C01810=1184.389,279.938,-67.679,-176.938,7.454,148.522
C01811=1184.393,279.690,-67.650,-176.940,7.452,148.522
C01812=1184.397,279.442,-67.621,-176.943,7.449,148.522
C01813=1184.402,279.194,-67.592,-176.946,7.446,148.522
C01814=1184.406,278.945,-67.564,-176.949,7.443,148.522
C01815=1184.410,278.696,-67.535,-176.951,7.441,148.523
C01816=1184.415,278.449,-67.506,-176.954,7.438,148.523
C01817=1184.419,278.200,-67.478,-176.957,7.435,148.523
C01818=1184.423,277.951,-67.449,-176.959,7.433,148.523
C01819=1184.428,277.704,-67.420,-176.962,7.430,148.523
C01820=1184.432,277.455,-67.392,-176.964,7.427,148.523
C01821=1184.437,277.207,-67.364,-176.967,7.425,148.523
C01822=1184.441,276.959,-67.335,-176.969,7.422,148.523
C01823=1184.445,276.710,-67.306,-176.972,7.419,148.523
C01824=1184.450,276.462,-67.278,-176.975,7.416,148.523
C01825=1184.454,276.214,-67.250,-176.977,7.413,148.523
C01826=1184.458,275.965,-67.220,-176.980,7.410,148.523
C01827=1184.462,275.717,-67.192,-176.982,7.407,148.523
C01828=1184.467,275.469,-67.164,-176.985,7.406,148.523
C01829=1184.471,275.221,-67.136,-176.988,7.403,148.523
C01830=1184.476,274.972,-67.107,-176.990,7.400,148.523
C01831=1184.480,274.724,-67.079,-176.993,7.398,148.524
C01832=1184.484,274.476,-67.050,-176.995,7.395,148.524
C01833=1184.488,274.227,-67.022,-176.998,7.392,148.524
C01834=1184.493,273.979,-66.993,-177.000,7.389,148.524
C01835=1184.497,273.730,-66.965,-177.003,7.386,148.524
C01836=1184.502,273.482,-66.937,-177.006,7.383,148.524
C01837=1184.506,273.233,-66.909,-177.008,7.381,148.524
C01838=1184.511,272.985,-66.880,-177.011,7.379,148.524
C01839=1184.515,272.737,-66.852,-177.014,7.376,148.524
C01840=1184.520,272.489,-66.824,-177.016,7.373,148.524
C01841=1184.523,272.241,-66.795,-177.019,7.370,148.524
C01842=1184.528,271.992,-66.766,-177.021,7.367,148.524
C01843=1184.532,271.744,-66.738,-177.023,7.365,148.524
C01844=1184.536,271.495,-66.710,-177.026,7.362,148.524
C01845=1184.541,271.247,-66.682,-177.029,7.359,148.525
C01846=1184.544,270.998,-66.654,-177.031,7.357,148.525
C01847=1184.550,270.750,-66.625,-177.034,7.354,148.525
C01848=1184.554,270.501,-66.598,-177.037,7.352,148.525
C01849=1184.559,270.253,-66.570,-177.039,7.349,148.525
C01850=1184.562,270.004,-66.541,-177.042,7.346,148.525
C01851=1184.567,269.756,-66.514,-177.045,7.343,148.525
C01852=1184.572,269.508,-66.485,-177.047,7.341,148.525
C01853=1184.576,269.260,-66.457,-177.049,7.338,148.525
C01854=1184.580,269.012,-66.429,-177.052,7.336,148.526
C01855=1184.584,268.763,-66.401,-177.055,7.333,148.526
C01856=1184.589,268.515,-66.373,-177.058,7.330,148.526
C01857=1184.593,268.266,-66.345,-177.060,7.328,148.526
C01858=1184.598,268.018,-66.317,-177.062,7.325,148.526
C01859=1184.602,267.769,-66.289,-177.065,7.322,148.526
C01860=1184.606,267.521,-66.261,-177.068,7.320,148.526
C01861=1184.611,267.273,-66.233,-177.071,7.317,148.526
C01862=1184.615,267.024,-66.205,-177.073,7.314,148.526
C01863=1184.620,266.776,-66.178,-177.075,7.312,148.526
C01864=1184.623,266.527,-66.149,-177.078,7.309,148.526
C01865=1184.628,266.279,-66.121,-177.080,7.307,148.526
C01866=1184.632,266.030,-66.094,-177.084,7.305,148.527
C01867=1184.637,265.782,-66.066,-177.086,7.302,148.527
C01868=1184.641,265.534,-66.038,-177.088,7.299,148.527
C01869=1184.646,265.285,-66.009,-177.091,7.296,148.527
C01870=1184.650,265.037,-65.982,-177.094,7.293,148.527
C01871=1184.655,264.789,-65.954,-177.096,7.291,148.527
C01872=1184.658,264.540,-65.926,-177.099,7.289,148.527
C01873=1184.664,264.292,-65.899,-177.101,7.286,148.527
C01874=1184.668,264.043,-65.871,-177.104,7.283,148.527
C01875=1184.672,263.795,-65.843,-177.107,7.280,148.527
C01876=1184.677,263.547,-65.816,-177.109,7.278,148.528
C01877=1184.680,263.298,-65.788,-177.112,7.276,148.528
C01878=1184.685,263.050,-65.761,-177.114,7.273,148.528
C01879=1184.690,262.777,-65.730,-177.117,7.270,148.528
C01880=1184.695,262.504,-65.700,-177.120,7.268,148.528
C01881=1184.700,262.231,-65.669,-177.123,7.265,148.528
C01882=1184.705,261.958,-65.639,-177.126,7.262,148.528
C01883=1184.709,261.710,-65.611,-177.129,7.259,148.528
C01884=1184.713,261.461,-65.583,-177.131,7.257,148.529
C01885=1184.718,261.213,-65.556,-177.134,7.254,148.529
C01886=1184.722,260.964,-65.528,-177.137,7.251,148.529
C01887=1184.727,260.716,-65.501,-177.139,7.249,148.529
C01888=1184.731,260.467,-65.473,-177.142,7.246,148.529
C01889=1184.735,260.219,-65.446,-177.144,7.244,148.529
C01890=1184.740,259.971,-65.418,-177.147,7.241,148.529
C01891=1184.744,259.722,-65.391,-177.149,7.239,148.529
C01892=1184.748,259.474,-65.363,-177.152,7.236,148.529
C01893=1184.753,259.225,-65.336,-177.155,7.233,148.530
C01894=1184.757,258.977,-65.309,-177.157,7.231,148.530
C01895=1184.761,258.728,-65.281,-177.160,7.228,148.530
C01896=1184.766,258.480,-65.254,-177.162,7.226,148.530
C01897=1184.770,258.231,-65.227,-177.165,7.223,148.530
C01898=1184.775,257.983,-65.199,-177.167,7.221,148.530
C01899=1184.779,257.734,-65.172,-177.170,7.218,148.530
C01900=1184.783,257.486,-65.145,-177.173,7.216,148.531
C01901=1184.788,257.238,-65.117,-177.175,7.213,148.531
C01902=1184.793,256.989,-65.090,-177.178,7.210,148.531
C01903=1184.797,256.740,-65.062,-177.180,7.208,148.531
C01904=1184.801,256.492,-65.035,-177.184,7.206,148.531
C01905=1184.806,256.244,-65.007,-177.186,7.203,148.531
C01906=1184.810,255.995,-64.980,-177.188,7.200,148.531
C01907=1184.815,255.747,-64.953,-177.191,7.197,148.531
C01908=1184.819,255.497,-64.926,-177.194,7.196,148.532
C01909=1184.823,255.250,-64.899,-177.197,7.193,148.532
C01910=1184.827,255.001,-64.872,-177.199,7.191,148.532
C01911=1184.832,254.753,-64.845,-177.202,7.188,148.532
C01912=1184.837,254.504,-64.818,-177.204,7.186,148.532
C01913=1184.841,254.256,-64.791,-177.207,7.183,148.532
C01914=1184.845,254.007,-64.763,-177.209,7.181,148.532
C01915=1184.850,253.758,-64.736,-177.212,7.178,148.533
C01916=1184.855,253.510,-64.709,-177.214,7.176,148.533
C01917=1184.858,253.262,-64.682,-177.217,7.173,148.533
C01918=1184.863,253.014,-64.655,-177.220,7.171,148.533
C01919=1184.867,252.765,-64.628,-177.222,7.168,148.533
C01920=1184.872,252.517,-64.601,-177.225,7.165,148.533
C01921=1184.876,252.267,-64.573,-177.228,7.163,148.533
C01922=1184.880,252.019,-64.547,-177.231,7.160,148.533
C01923=1184.885,251.771,-64.520,-177.233,7.158,148.534
C01924=1184.889,251.522,-64.493,-177.236,7.155,148.534
C01925=1184.894,251.274,-64.466,-177.238,7.153,148.534
C01926=1184.898,251.026,-64.439,-177.241,7.150,148.534
C01927=1184.903,250.777,-64.412,-177.243,7.148,148.534
C01928=1184.907,250.529,-64.385,-177.246,7.145,148.534
C01929=1184.912,250.280,-64.358,-177.248,7.143,148.534
C01930=1184.915,250.031,-64.331,-177.252,7.141,148.535
C01931=1184.920,249.783,-64.304,-177.254,7.138,148.535
C01932=1184.925,249.534,-64.278,-177.256,7.135,148.535
C01933=1184.930,249.285,-64.251,-177.259,7.134,148.535
C01934=1184.933,249.037,-64.224,-177.262,7.131,148.535
C01935=1184.938,248.788,-64.197,-177.264,7.129,148.535
C01936=1184.943,248.540,-64.170,-177.267,7.126,148.536
C01937=1184.947,248.292,-64.144,-177.269,7.124,148.536
C01938=1184.951,248.043,-64.116,-177.272,7.121,148.536
C01939=1184.956,247.794,-64.090,-177.275,7.119,148.536
C01940=1184.960,247.546,-64.064,-177.278,7.116,148.536
C01941=1184.965,247.298,-64.037,-177.280,7.114,148.536
C01942=1184.969,247.049,-64.010,-177.283,7.111,148.537
C01943=1184.973,246.801,-63.983,-177.285,7.109,148.537
C01944=1184.978,246.552,-63.957,-177.288,7.106,148.537
C01945=1184.982,246.304,-63.930,-177.290,7.104,148.537
C01946=1184.987,246.055,-63.903,-177.293,7.101,148.537
C01947=1184.991,245.806,-63.877,-177.296,7.099,148.537
C01948=1184.996,245.558,-63.850,-177.299,7.096,148.537
C01949=1185.001,245.309,-63.823,-177.301,7.094,148.538
C01950=1185.004,245.061,-63.797,-177.304,7.092,148.538
C01951=1185.009,244.812,-63.770,-177.306,7.089,148.538
C01952=1185.013,244.564,-63.744,-177.309,7.088,148.538
C01953=1185.018,244.315,-63.717,-177.311,7.085,148.538
C01954=1185.022,244.066,-63.691,-177.314,7.082,148.538
C01955=1185.027,243.818,-63.664,-177.317,7.080,148.539
C01956=1185.031,243.569,-63.638,-177.319,7.078,148.539
C01957=1185.036,243.321,-63.611,-177.322,7.075,148.539
C01958=1185.040,243.072,-63.585,-177.324,7.073,148.539
C01959=1185.045,242.823,-63.559,-177.327,7.070,148.539
C01960=1185.049,242.575,-63.532,-177.330,7.068,148.540
C01961=1185.054,242.326,-63.506,-177.333,7.065,148.540
C01962=1185.057,242.078,-63.479,-177.335,7.063,148.540
C01963=1185.062,241.829,-63.453,-177.338,7.060,148.540
C01964=1185.067,241.581,-63.427,-177.341,7.058,148.540
C01965=1185.072,241.332,-63.400,-177.343,7.056,148.540
C01966=1185.076,241.084,-63.374,-177.345,7.053,148.540
C01967=1185.081,240.835,-63.348,-177.348,7.052,148.541
C01968=1185.085,240.587,-63.321,-177.351,7.049,148.541
C01969=1185.089,240.338,-63.295,-177.353,7.047,148.541
C01970=1185.094,240.089,-63.268,-177.356,7.044,148.541
C01971=1185.098,239.841,-63.243,-177.359,7.042,148.542
C01972=1185.102,239.592,-63.216,-177.362,7.039,148.542
C01973=1185.107,239.344,-63.190,-177.364,7.037,148.542
C01974=1185.112,239.095,-63.164,-177.366,7.035,148.542
C01975=1185.116,238.847,-63.137,-177.369,7.032,148.542
C01976=1185.120,238.598,-63.112,-177.372,7.030,148.542
C01977=1185.125,238.349,-63.086,-177.375,7.027,148.543
C01978=1185.129,238.101,-63.059,-177.377,7.025,148.543
C01979=1185.134,237.852,-63.033,-177.380,7.022,148.543
C01980=1185.138,237.604,-63.008,-177.383,7.021,148.543
C01981=1185.143,237.355,-62.981,-177.385,7.018,148.543
C01982=1185.147,237.106,-62.955,-177.388,7.016,148.544
C01983=1185.152,236.835,-62.926,-177.391,7.013,148.544
C01984=1185.157,236.563,-62.897,-177.393,7.011,148.544
C01985=1185.162,236.292,-62.870,-177.397,7.008,148.544
C01986=1185.167,236.020,-62.841,-177.399,7.005,148.544
C01987=1185.171,235.772,-62.815,-177.402,7.004,148.545
C01988=1185.176,235.522,-62.789,-177.404,7.001,148.545
C01989=1185.180,235.274,-62.762,-177.407,6.999,148.545
C01990=1185.185,235.026,-62.737,-177.409,6.997,148.545
C01991=1185.189,234.777,-62.711,-177.413,6.994,148.545
C01992=1185.194,234.528,-62.685,-177.415,6.992,148.546
C01993=1185.198,234.279,-62.659,-177.418,6.989,148.546
C01994=1185.202,234.031,-62.633,-177.420,6.987,148.546
C01995=1185.207,233.783,-62.607,-177.423,6.985,148.546
C01996=1185.211,233.534,-62.582,-177.426,6.982,148.546
C01997=1185.216,233.285,-62.555,-177.428,6.980,148.547
C01998=1185.220,233.036,-62.530,-177.430,6.978,148.547
C01999=1185.225,232.788,-62.504,-177.434,6.976,148.547
C02000=1185.229,232.540,-62.478,-177.436,6.974,148.547
C02001=1185.233,232.291,-62.453,-177.439,6.971,148.547
C02002=1185.238,232.043,-62.427,-177.441,6.969,148.548
C02003=1185.243,231.794,-62.401,-177.444,6.967,148.548
C02004=1185.247,231.545,-62.375,-177.447,6.964,148.548
C02005=1185.252,231.296,-62.349,-177.449,6.962,148.548
C02006=1185.257,231.048,-62.324,-177.452,6.959,148.548
C02007=1185.261,230.799,-62.298,-177.455,6.957,148.549
C02008=1185.265,230.550,-62.273,-177.457,6.955,148.549
C02009=1185.270,230.302,-62.247,-177.460,6.953,148.549
C02010=1185.274,230.053,-62.221,-177.463,6.951,148.549
C02011=1185.278,229.804,-62.196,-177.465,6.949,148.550
C02012=1185.282,229.556,-62.170,-177.468,6.946,148.550
C02013=1185.287,229.308,-62.144,-177.470,6.944,148.550
C02014=1185.292,229.059,-62.119,-177.473,6.942,148.550
C02015=1185.297,228.810,-62.092,-177.476,6.939,148.550
C02016=1185.301,228.562,-62.067,-177.478,6.937,148.551
C02017=1185.306,228.312,-62.042,-177.481,6.934,148.551
C02018=1185.311,228.064,-62.017,-177.484,6.932,148.551
C02019=1185.315,227.815,-61.991,-177.486,6.931,148.551
C02020=1185.319,227.566,-61.965,-177.489,6.928,148.551
C02021=1185.324,227.318,-61.940,-177.492,6.926,148.552
C02022=1185.328,227.069,-61.914,-177.494,6.924,148.552
C02023=1185.333,226.820,-61.889,-177.497,6.921,148.552
C02024=1185.338,226.572,-61.864,-177.499,6.919,148.552
C02025=1185.342,226.323,-61.838,-177.502,6.917,148.553
C02026=1185.346,226.074,-61.812,-177.505,6.914,148.553
C02027=1185.350,225.827,-61.787,-177.507,6.912,148.553
C02028=1185.355,225.577,-61.762,-177.510,6.910,148.553
C02029=1185.359,225.329,-61.737,-177.513,6.907,148.553
C02030=1185.364,225.080,-61.711,-177.515,6.906,148.554
C02031=1185.368,224.831,-61.686,-177.518,6.904,148.554
C02032=1185.373,224.583,-61.661,-177.521,6.901,148.554
C02033=1185.377,224.334,-61.635,-177.523,6.899,148.555
C02034=1185.382,224.085,-61.610,-177.526,6.897,148.555
C02035=1185.387,223.836,-61.584,-177.529,6.894,148.555
C02036=1185.391,223.588,-61.559,-177.531,6.892,148.555
C02037=1185.396,223.339,-61.534,-177.534,6.890,148.555
C02038=1185.400,223.091,-61.509,-177.537,6.888,148.556
C02039=1185.404,222.842,-61.484,-177.539,6.886,148.556
C02040=1185.409,222.593,-61.458,-177.542,6.884,148.556
C02041=1185.414,222.345,-61.433,-177.545,6.881,148.556
C02042=1185.418,222.095,-61.408,-177.547,6.879,148.557
C02043=1185.423,221.847,-61.383,-177.550,6.877,148.557
C02044=1185.426,221.599,-61.358,-177.552,6.874,148.557
C02045=1185.432,221.350,-61.333,-177.555,6.872,148.557
C02046=1185.436,221.101,-61.307,-177.558,6.871,148.558
C02047=1185.441,220.852,-61.282,-177.560,6.868,148.558
C02048=1185.445,220.604,-61.257,-177.563,6.866,148.558
C02049=1185.450,220.355,-61.233,-177.566,6.864,148.558
C02050=1185.454,220.106,-61.207,-177.568,6.862,148.558
C02051=1185.459,219.858,-61.182,-177.571,6.859,148.559
C02052=1185.463,219.609,-61.156,-177.574,6.857,148.559
C02053=1185.468,219.360,-61.132,-177.576,6.855,148.559
C02054=1185.472,219.111,-61.107,-177.579,6.853,148.560
C02055=1185.477,218.863,-61.082,-177.582,6.851,148.560
C02056=1185.481,218.614,-61.057,-177.584,6.849,148.560
C02057=1185.486,218.366,-61.032,-177.587,6.846,148.560
C02058=1185.490,218.116,-61.007,-177.589,6.844,148.560
C02059=1185.495,217.868,-60.982,-177.592,6.842,148.561
C02060=1185.499,217.620,-60.958,-177.595,6.840,148.561
C02061=1185.504,217.370,-60.933,-177.598,6.837,148.561
C02062=1185.509,217.122,-60.908,-177.600,6.835,148.561
C02063=1185.512,216.873,-60.883,-177.603,6.834,148.562
C02064=1185.518,216.624,-60.858,-177.606,6.831,148.562
C02065=1185.522,216.375,-60.833,-177.608,6.829,148.562
C02066=1185.526,216.127,-60.808,-177.611,6.827,148.563
C02067=1185.531,215.878,-60.784,-177.613,6.825,148.563
C02068=1185.536,215.629,-60.759,-177.616,6.822,148.563
C02069=1185.540,215.381,-60.734,-177.619,6.820,148.563
C02070=1185.544,215.132,-60.709,-177.622,6.819,148.564
C02071=1185.549,214.883,-60.685,-177.624,6.816,148.564
C02072=1185.554,214.635,-60.660,-177.627,6.814,148.564
C02073=1185.559,214.385,-60.635,-177.630,6.812,148.564
C02074=1185.563,214.137,-60.610,-177.632,6.810,148.565
C02075=1185.567,213.888,-60.585,-177.635,6.807,148.565
C02076=1185.572,213.640,-60.561,-177.638,6.806,148.565
C02077=1185.577,213.391,-60.536,-177.640,6.803,148.565
C02078=1185.580,213.142,-60.512,-177.643,6.802,148.566
C02079=1185.586,212.893,-60.487,-177.646,6.799,148.566
C02080=1185.590,212.645,-60.462,-177.648,6.797,148.566
C02081=1185.594,212.396,-60.437,-177.651,6.795,148.566
C02082=1185.599,212.147,-60.413,-177.653,6.793,148.567
C02083=1185.604,211.899,-60.389,-177.656,6.791,148.567
C02084=1185.608,211.649,-60.364,-177.659,6.788,148.567
C02085=1185.613,211.401,-60.340,-177.661,6.787,148.568
C02086=1185.618,211.152,-60.315,-177.664,6.785,148.568
C02087=1185.622,210.882,-60.288,-177.667,6.782,148.568
C02088=1185.627,210.611,-60.262,-177.669,6.780,148.568
C02089=1185.632,210.341,-60.235,-177.673,6.777,148.569
C02090=1185.637,210.070,-60.209,-177.676,6.775,148.569
C02091=1185.641,209.821,-60.185,-177.678,6.773,148.569
C02092=1185.646,209.573,-60.160,-177.681,6.771,148.570
C02093=1185.651,209.324,-60.136,-177.683,6.769,148.570
C02094=1185.655,209.075,-60.111,-177.686,6.767,148.570
C02095=1185.660,208.826,-60.087,-177.689,6.765,148.570
C02096=1185.665,208.578,-60.062,-177.692,6.763,148.571
C02097=1185.669,208.329,-60.038,-177.694,6.761,148.571
C02098=1185.673,208.080,-60.014,-177.697,6.759,148.571
C02099=1185.678,207.831,-59.989,-177.700,6.756,148.571
C02100=1185.682,207.583,-59.965,-177.703,6.754,148.572
C02101=1185.688,207.334,-59.940,-177.705,6.752,148.572
C02102=1185.691,207.085,-59.916,-177.707,6.750,148.572
C02103=1185.696,206.836,-59.892,-177.710,6.749,148.573
C02104=1185.701,206.587,-59.868,-177.713,6.746,148.573
C02105=1185.706,206.339,-59.844,-177.716,6.744,148.573
C02106=1185.709,206.090,-59.819,-177.718,6.742,148.573
C02107=1185.715,205.841,-59.794,-177.721,6.740,148.574
C02108=1185.719,205.592,-59.771,-177.724,6.737,148.574
C02109=1185.724,205.344,-59.747,-177.726,6.736,148.574
C02110=1185.729,205.095,-59.722,-177.729,6.734,148.574
C02111=1185.733,204.846,-59.698,-177.732,6.732,148.575
C02112=1185.737,204.597,-59.674,-177.734,6.730,148.575
C02113=1185.742,204.348,-59.651,-177.737,6.727,148.575
C02114=1185.747,204.100,-59.626,-177.740,6.725,148.576
C02115=1185.751,203.851,-59.602,-177.742,6.724,148.576
C02116=1185.755,203.602,-59.578,-177.745,6.722,148.576
C02117=1185.760,203.353,-59.554,-177.747,6.720,148.576
C02118=1185.765,203.104,-59.529,-177.750,6.717,148.577
C02119=1185.769,202.856,-59.505,-177.753,6.715,148.577
C02120=1185.774,202.607,-59.482,-177.756,6.713,148.577
C02121=1185.778,202.359,-59.458,-177.758,6.711,148.578
C02122=1185.782,202.109,-59.434,-177.761,6.709,148.578
C02123=1185.788,201.860,-59.409,-177.764,6.707,148.578
C02124=1185.792,201.612,-59.385,-177.766,6.705,148.579
C02125=1185.797,201.363,-59.362,-177.769,6.703,148.579
C02126=1185.801,201.114,-59.338,-177.771,6.701,148.579
C02127=1185.806,200.865,-59.315,-177.774,6.699,148.579
C02128=1185.811,200.617,-59.290,-177.777,6.698,148.580
C02129=1185.815,200.368,-59.266,-177.780,6.695,148.580
C02130=1185.819,200.118,-59.242,-177.782,6.693,148.580
C02131=1185.824,199.870,-59.218,-177.785,6.691,148.581
C02132=1185.828,199.621,-59.195,-177.787,6.689,148.581
C02133=1185.833,199.373,-59.171,-177.790,6.687,148.581
C02134=1185.838,199.123,-59.147,-177.793,6.686,148.582
C02135=1185.842,198.875,-59.123,-177.796,6.683,148.582
C02136=1185.847,198.626,-59.099,-177.798,6.681,148.582
C02137=1185.852,198.377,-59.075,-177.801,6.679,148.582
C02138=1185.856,198.128,-59.052,-177.803,6.677,148.583
C02139=1185.861,197.880,-59.028,-177.806,6.675,148.583
C02140=1185.866,197.631,-59.004,-177.809,6.674,148.583
C02141=1185.870,197.382,-58.981,-177.811,6.671,148.583
C02142=1185.874,197.133,-58.956,-177.814,6.669,148.584
C02143=1185.879,196.884,-58.933,-177.817,6.667,148.584
C02144=1185.883,196.635,-58.909,-177.819,6.665,148.585
C02145=1185.888,196.386,-58.886,-177.822,6.663,148.585
C02146=1185.893,196.137,-58.862,-177.825,6.662,148.585
C02147=1185.897,195.889,-58.838,-177.827,6.660,148.585
C02148=1185.902,195.640,-58.815,-177.830,6.657,148.586
C02149=1185.906,195.391,-58.792,-177.833,6.655,148.586
C02150=1185.911,195.142,-58.767,-177.836,6.653,148.586
C02151=1185.915,194.893,-58.744,-177.838,6.652,148.587
C02152=1185.920,194.644,-58.721,-177.841,6.650,148.587
C02153=1185.925,194.395,-58.697,-177.843,6.648,148.587
C02154=1185.929,194.147,-58.673,-177.846,6.646,148.588
C02155=1185.934,193.898,-58.650,-177.848,6.644,148.588
C02156=1185.939,193.649,-58.627,-177.852,6.641,148.588
C02157=1185.943,193.400,-58.603,-177.854,6.640,148.589
C02158=1185.948,193.151,-58.579,-177.857,6.638,148.589
C02159=1185.952,192.902,-58.556,-177.859,6.636,148.589
C02160=1185.957,192.653,-58.532,-177.862,6.634,148.589
C02161=1185.962,192.404,-58.509,-177.864,6.632,148.590
C02162=1185.966,192.155,-58.486,-177.867,6.630,148.590
C02163=1185.971,191.908,-58.463,-177.870,6.628,148.590
C02164=1185.975,191.659,-58.439,-177.873,6.626,148.591
C02165=1185.980,191.410,-58.416,-177.876,6.624,148.591
C02166=1185.985,191.161,-58.393,-177.878,6.622,148.591
C02167=1185.990,190.912,-58.369,-177.881,6.620,148.592
C02168=1185.994,190.663,-58.346,-177.883,6.618,148.592
C02169=1185.999,190.414,-58.322,-177.886,6.617,148.592
C02170=1186.003,190.165,-58.300,-177.889,6.615,148.593
C02171=1186.007,189.916,-58.276,-177.891,6.613,148.593
C02172=1186.012,189.667,-58.252,-177.894,6.611,148.593
C02173=1186.017,189.418,-58.229,-177.897,6.608,148.593
C02174=1186.021,189.169,-58.206,-177.899,6.606,148.594
C02175=1186.027,188.921,-58.183,-177.902,6.605,148.594
C02176=1186.031,188.672,-58.160,-177.905,6.603,148.595
C02177=1186.035,188.423,-58.136,-177.907,6.601,148.595
C02178=1186.040,188.174,-58.113,-177.910,6.599,148.595
C02179=1186.045,187.925,-58.090,-177.913,6.597,148.596
C02180=1186.049,187.676,-58.067,-177.915,6.596,148.596
C02181=1186.053,187.427,-58.044,-177.918,6.594,148.596
C02182=1186.058,187.178,-58.020,-177.920,6.592,148.596
C02183=1186.063,186.930,-57.997,-177.923,6.590,148.597
C02184=1186.067,186.681,-57.974,-177.925,6.588,148.597
C02185=1186.072,186.432,-57.952,-177.929,6.586,148.597
C02186=1186.077,186.183,-57.928,-177.931,6.584,148.598
C02187=1186.082,185.934,-57.905,-177.934,6.582,148.598
C02188=1186.086,185.685,-57.882,-177.937,6.580,148.599
C02189=1186.091,185.437,-57.859,-177.939,6.578,148.599
C02190=1186.096,185.188,-57.836,-177.942,6.577,148.599
C02191=1186.100,184.918,-57.812,-177.945,6.575,148.600
C02192=1186.106,184.648,-57.787,-177.948,6.572,148.600
C02193=1186.111,184.379,-57.761,-177.951,6.570,148.600
C02194=1186.116,184.109,-57.737,-177.953,6.569,148.601
C02195=1186.120,183.860,-57.714,-177.956,6.567,148.601
C02196=1186.125,183.611,-57.690,-177.959,6.565,148.601
C02197=1186.129,183.362,-57.668,-177.961,6.563,148.602
C02198=1186.135,183.113,-57.645,-177.964,6.561,148.602
C02199=1186.138,182.865,-57.623,-177.966,6.559,148.602
C02200=1186.143,182.616,-57.599,-177.969,6.557,148.603
C02201=1186.148,182.367,-57.576,-177.972,6.555,148.603
C02202=1186.152,182.117,-57.554,-177.975,6.553,148.603
C02203=1186.157,181.869,-57.531,-177.977,6.551,148.604
C02204=1186.161,181.620,-57.508,-177.980,6.550,148.604
C02205=1186.166,181.371,-57.485,-177.983,6.548,148.604
C02206=1186.170,181.122,-57.463,-177.985,6.546,148.605
C02207=1186.176,180.873,-57.440,-177.988,6.544,148.605
C02208=1186.181,180.624,-57.417,-177.991,6.542,148.605
C02209=1186.185,180.375,-57.394,-177.993,6.541,148.606
C02210=1186.189,180.126,-57.371,-177.996,6.539,148.606
C02211=1186.194,179.877,-57.349,-177.999,6.537,148.606
C02212=1186.199,179.628,-57.326,-178.001,6.535,148.607
C02213=1186.203,179.380,-57.303,-178.004,6.533,148.607
C02214=1186.208,179.131,-57.281,-178.006,6.531,148.607
C02215=1186.212,178.882,-57.258,-178.009,6.530,148.608
C02216=1186.217,178.632,-57.235,-178.012,6.528,148.608
C02217=1186.221,178.384,-57.213,-178.014,6.526,148.608
C02218=1186.227,178.135,-57.190,-178.017,6.524,148.609
C02219=1186.231,177.886,-57.168,-178.020,6.522,148.609
C02220=1186.236,177.637,-57.144,-178.022,6.521,148.610
C02221=1186.241,177.388,-57.123,-178.025,6.519,148.610
C02222=1186.245,177.140,-57.100,-178.028,6.517,148.610
C02223=1186.250,176.890,-57.077,-178.030,6.515,148.611
C02224=1186.254,176.642,-57.055,-178.033,6.514,148.611
C02225=1186.259,176.392,-57.032,-178.036,6.512,148.611
C02226=1186.263,176.143,-57.010,-178.038,6.510,148.612
C02227=1186.269,175.895,-56.987,-178.041,6.508,148.612
C02228=1186.273,175.645,-56.965,-178.044,6.506,148.612
C02229=1186.277,175.396,-56.942,-178.046,6.505,148.613
C02230=1186.283,175.148,-56.920,-178.049,6.503,148.613
C02231=1186.286,174.899,-56.897,-178.052,6.501,148.613
C02232=1186.292,174.650,-56.875,-178.054,6.499,148.614
C02233=1186.296,174.401,-56.853,-178.057,6.497,148.614
C02234=1186.300,174.152,-56.830,-178.060,6.496,148.615
C02235=1186.306,173.903,-56.808,-178.062,6.494,148.615
C02236=1186.310,173.654,-56.786,-178.065,6.492,148.615
C02237=1186.315,173.406,-56.763,-178.068,6.490,148.616
C02238=1186.320,173.156,-56.741,-178.071,6.489,148.616
C02239=1186.324,172.906,-56.719,-178.073,6.487,148.616
C02240=1186.329,172.658,-56.696,-178.076,6.485,148.617
C02241=1186.334,172.409,-56.674,-178.079,6.483,148.617
C02242=1186.338,172.160,-56.652,-178.081,6.481,148.617
C02243=1186.342,171.911,-56.629,-178.084,6.480,148.618
C02244=1186.347,171.663,-56.607,-178.087,6.478,148.618
C02245=1186.352,171.413,-56.585,-178.089,6.476,148.619
C02246=1186.357,171.164,-56.563,-178.092,6.474,148.619
C02247=1186.361,170.915,-56.541,-178.095,6.473,148.619
C02248=1186.366,170.666,-56.518,-178.097,6.471,148.620
C02249=1186.371,170.418,-56.496,-178.100,6.469,148.620
C02250=1186.375,170.168,-56.474,-178.103,6.467,148.620
C02251=1186.380,169.920,-56.452,-178.105,6.465,148.621
C02252=1186.384,169.670,-56.430,-178.108,6.464,148.621
C02253=1186.390,169.422,-56.407,-178.111,6.462,148.621
C02254=1186.394,169.173,-56.385,-178.113,6.460,148.622
C02255=1186.399,168.924,-56.364,-178.116,6.458,148.622
C02256=1186.403,168.675,-56.342,-178.119,6.457,148.623
C02257=1186.409,168.426,-56.319,-178.121,6.455,148.623
C02258=1186.413,168.176,-56.297,-178.124,6.453,148.623
C02259=1186.418,167.928,-56.276,-178.126,6.452,148.624
C02260=1186.422,167.678,-56.253,-178.129,6.450,148.624
C02261=1186.427,167.430,-56.232,-178.131,6.448,148.624
C02262=1186.431,167.181,-56.209,-178.134,6.447,148.625
C02263=1186.437,166.932,-56.187,-178.137,6.445,148.625
C02264=1186.441,166.683,-56.165,-178.140,6.443,148.626
C02265=1186.446,166.434,-56.143,-178.142,6.441,148.626
C02266=1186.450,166.185,-56.121,-178.145,6.440,148.626
C02267=1186.455,165.936,-56.099,-178.148,6.438,148.627
C02268=1186.459,165.687,-56.077,-178.150,6.436,148.627
C02269=1186.464,165.438,-56.056,-178.153,6.434,148.627
C02270=1186.468,165.189,-56.034,-178.156,6.432,148.628
C02271=1186.473,164.940,-56.012,-178.158,6.431,148.628
C02272=1186.478,164.691,-55.990,-178.161,6.429,148.628
C02273=1186.482,164.442,-55.968,-178.164,6.427,148.629
C02274=1186.488,164.192,-55.947,-178.166,6.425,148.629
C02275=1186.492,163.943,-55.924,-178.168,6.424,148.630
C02276=1186.497,163.695,-55.903,-178.172,6.423,148.630
C02277=1186.502,163.445,-55.881,-178.174,6.421,148.631
C02278=1186.506,163.197,-55.859,-178.177,6.419,148.631
C02279=1186.511,162.948,-55.837,-178.180,6.418,148.631
C02280=1186.516,162.699,-55.815,-178.182,6.416,148.632
C02281=1186.520,162.450,-55.794,-178.185,6.414,148.632
C02282=1186.525,162.201,-55.772,-178.188,6.412,148.632
C02283=1186.530,161.951,-55.751,-178.190,6.410,148.633
C02284=1186.535,161.703,-55.729,-178.193,6.409,148.633
C02285=1186.539,161.453,-55.707,-178.196,6.407,148.634
C02286=1186.544,161.205,-55.685,-178.198,6.406,148.634
C02287=1186.549,160.956,-55.664,-178.200,6.404,148.634
C02288=1186.553,160.706,-55.642,-178.203,6.402,148.635
C02289=1186.558,160.457,-55.621,-178.206,6.401,148.635
C02290=1186.562,160.208,-55.599,-178.209,6.399,148.635
C02291=1186.567,159.960,-55.577,-178.212,6.397,148.636
C02292=1186.572,159.711,-55.556,-178.214,6.396,148.636
C02293=1186.576,159.461,-55.534,-178.217,6.394,148.637
C02294=1186.581,159.213,-55.513,-178.220,6.392,148.637
C02295=1186.586,158.943,-55.489,-178.222,6.390,148.638
C02296=1186.591,158.674,-55.467,-178.225,6.389,148.638
C02297=1186.596,158.405,-55.443,-178.228,6.387,148.638
C02298=1186.601,158.136,-55.420,-178.231,6.385,148.639
C02299=1186.606,157.888,-55.398,-178.234,6.384,148.639
C02300=1186.611,157.638,-55.377,-178.236,6.382,148.640
C02301=1186.615,157.389,-55.355,-178.239,6.380,148.640
C02302=1186.620,157.140,-55.333,-178.242,6.378,148.640
C02303=1186.625,156.891,-55.312,-178.244,6.377,148.641
C02304=1186.630,156.643,-55.291,-178.246,6.376,148.641
C02305=1186.634,156.393,-55.270,-178.249,6.374,148.641
C02306=1186.639,156.144,-55.248,-178.252,6.372,148.642
C02307=1186.644,155.895,-55.227,-178.255,6.371,148.642
C02308=1186.648,155.646,-55.205,-178.258,6.369,148.643
C02309=1186.653,155.397,-55.184,-178.260,6.367,148.643
C02310=1186.658,155.148,-55.163,-178.263,6.365,148.644
C02311=1186.663,154.899,-55.142,-178.265,6.364,148.644
C02312=1186.667,154.649,-55.120,-178.268,6.363,148.644
C02313=1186.672,154.401,-55.099,-178.271,6.361,148.645
C02314=1186.676,154.152,-55.078,-178.273,6.359,148.645
C02315=1186.681,153.903,-55.056,-178.276,6.358,148.646
C02316=1186.686,153.653,-55.035,-178.279,6.356,148.646
C02317=1186.691,153.405,-55.013,-178.282,6.354,148.646
C02318=1186.695,153.156,-54.993,-178.284,6.353,148.647
C02319=1186.700,152.906,-54.972,-178.287,6.351,148.647
C02320=1186.705,152.658,-54.950,-178.289,6.350,148.648
C02321=1186.710,152.408,-54.929,-178.292,6.348,148.648
C02322=1186.714,152.159,-54.908,-178.295,6.346,148.648
C02323=1186.719,151.910,-54.887,-178.298,6.345,148.649
C02324=1186.724,151.662,-54.865,-178.300,6.344,148.649
C02325=1186.728,151.413,-54.845,-178.303,6.342,148.650
C02326=1186.733,151.163,-54.824,-178.305,6.340,148.650
C02327=1186.738,150.914,-54.802,-178.308,6.338,148.650
C02328=1186.742,150.665,-54.782,-178.311,6.337,148.651
C02329=1186.748,150.416,-54.761,-178.313,6.335,148.651
C02330=1186.752,150.167,-54.739,-178.316,6.334,148.652
C02331=1186.757,149.918,-54.719,-178.319,6.332,148.652
C02332=1186.761,149.668,-54.697,-178.321,6.331,148.653
C02333=1186.766,149.420,-54.676,-178.324,6.329,148.653
C02334=1186.771,149.171,-54.655,-178.327,6.327,148.653
C02335=1186.776,148.921,-54.634,-178.329,6.325,148.654
C02336=1186.781,148.672,-54.613,-178.331,6.324,148.654
C02337=1186.785,148.424,-54.592,-178.335,6.323,148.655
C02338=1186.790,148.175,-54.571,-178.337,6.321,148.655
C02339=1186.794,147.925,-54.550,-178.340,6.319,148.656
C02340=1186.799,147.676,-54.530,-178.343,6.318,148.656
C02341=1186.804,147.427,-54.508,-178.345,6.317,148.656
C02342=1186.809,147.178,-54.487,-178.347,6.315,148.657
C02343=1186.814,146.929,-54.466,-178.351,6.314,148.657
C02344=1186.818,146.680,-54.446,-178.353,6.312,148.658
C02345=1186.823,146.431,-54.425,-178.356,6.310,148.658
C02346=1186.828,146.182,-54.405,-178.359,6.308,148.658
C02347=1186.833,145.933,-54.383,-178.361,6.307,148.659
C02348=1186.837,145.684,-54.363,-178.364,6.306,148.659
C02349=1186.842,145.434,-54.341,-178.367,6.304,148.660
C02350=1186.846,145.185,-54.321,-178.369,6.302,148.660
C02351=1186.851,144.936,-54.300,-178.371,6.301,148.661
C02352=1186.856,144.687,-54.280,-178.374,6.300,148.661
C02353=1186.861,144.438,-54.259,-178.377,6.298,148.661
C02354=1186.865,144.189,-54.238,-178.380,6.296,148.662
C02355=1186.871,143.939,-54.217,-178.383,6.295,148.662
C02356=1186.875,143.691,-54.197,-178.385,6.294,148.663
C02357=1186.880,143.441,-54.176,-178.388,6.292,148.663
C02358=1186.884,143.193,-54.155,-178.390,6.290,148.664
C02359=1186.890,142.944,-54.134,-178.393,6.289,148.664
C02360=1186.894,142.695,-54.114,-178.396,6.287,148.664
C02361=1186.898,142.446,-54.093,-178.398,6.286,148.665
C02362=1186.904,142.197,-54.072,-178.401,6.284,148.665
C02363=1186.908,141.948,-54.052,-178.404,6.283,148.666
C02364=1186.914,141.698,-54.032,-178.406,6.281,148.666
C02365=1186.918,141.449,-54.011,-178.409,6.280,148.667
C02366=1186.922,141.200,-53.991,-178.412,6.279,148.667
C02367=1186.928,140.951,-53.970,-178.414,6.277,148.667
C02368=1186.932,140.702,-53.950,-178.417,6.275,148.668
C02369=1186.937,140.452,-53.929,-178.419,6.274,148.668
C02370=1186.942,140.203,-53.908,-178.422,6.273,148.669
C02371=1186.946,139.954,-53.888,-178.425,6.271,148.669
C02372=1186.951,139.705,-53.867,-178.428,6.269,148.670
C02373=1186.956,139.456,-53.847,-178.430,6.267,148.670
C02374=1186.960,139.207,-53.826,-178.432,6.266,148.670
C02375=1186.966,138.957,-53.806,-178.436,6.265,148.671
C02376=1186.970,138.708,-53.786,-178.438,6.263,148.671
C02377=1186.974,138.460,-53.765,-178.441,6.261,148.672
C02378=1186.980,138.210,-53.744,-178.443,6.261,148.672
C02379=1186.984,137.961,-53.724,-178.446,6.259,148.673
C02380=1186.988,137.712,-53.703,-178.449,6.257,148.673
C02381=1186.994,137.462,-53.683,-178.452,6.256,148.674
C02382=1186.998,137.214,-53.663,-178.454,6.255,148.674
C02383=1187.003,136.965,-53.642,-178.456,6.253,148.674
C02384=1187.007,136.716,-53.622,-178.460,6.251,148.675
C02385=1187.013,136.466,-53.602,-178.462,6.251,148.675
C02386=1187.017,136.217,-53.581,-178.464,6.249,148.676
C02387=1187.022,135.969,-53.561,-178.467,6.247,148.676
C02388=1187.027,135.720,-53.541,-178.470,6.246,148.677
C02389=1187.032,135.470,-53.521,-178.472,6.245,148.677
C02390=1187.037,135.221,-53.500,-178.475,6.243,148.678
C02391=1187.041,134.972,-53.480,-178.478,6.241,148.678
C02392=1187.046,134.722,-53.460,-178.481,6.240,148.679
C02393=1187.050,134.473,-53.440,-178.483,6.239,148.679
C02394=1187.055,134.224,-53.419,-178.486,6.237,148.679
C02395=1187.060,133.974,-53.399,-178.489,6.235,148.680
C02396=1187.065,133.726,-53.379,-178.491,6.234,148.680
C02397=1187.070,133.477,-53.359,-178.494,6.233,148.681
C02398=1187.074,133.228,-53.339,-178.496,6.231,148.681
C02399=1187.080,132.959,-53.317,-178.499,6.229,148.682
C02400=1187.085,132.691,-53.296,-178.502,6.228,148.682
C02401=1187.090,132.422,-53.274,-178.505,6.226,148.683
C02402=1187.095,132.154,-53.252,-178.508,6.225,148.683
C02403=1187.100,131.904,-53.232,-178.510,6.224,148.684
C02404=1187.105,131.655,-53.212,-178.513,6.222,148.684
C02405=1187.110,131.405,-53.192,-178.516,6.220,148.684
C02406=1187.114,131.156,-53.172,-178.518,6.220,148.685
C02407=1187.119,130.908,-53.152,-178.521,6.218,148.685
C02408=1187.124,130.659,-53.132,-178.524,6.216,148.686
C02409=1187.128,130.409,-53.112,-178.527,6.215,148.686
C02410=1187.133,130.160,-53.092,-178.529,6.214,148.687
C02411=1187.138,129.910,-53.072,-178.532,6.212,148.687
C02412=1187.143,129.662,-53.052,-178.534,6.210,148.688
C02413=1187.148,129.412,-53.032,-178.537,6.210,148.688
C02414=1187.153,129.163,-53.012,-178.540,6.208,148.689
C02415=1187.157,128.914,-52.992,-178.542,6.206,148.689
C02416=1187.162,128.665,-52.972,-178.545,6.205,148.689
C02417=1187.167,128.416,-52.952,-178.548,6.204,148.690
C02418=1187.172,128.166,-52.933,-178.550,6.202,148.690
C02419=1187.176,127.918,-52.912,-178.553,6.201,148.691
C02420=1187.181,127.668,-52.893,-178.556,6.200,148.691
C02421=1187.186,127.420,-52.873,-178.558,6.198,148.692
C02422=1187.191,127.170,-52.853,-178.561,6.197,148.692
C02423=1187.196,126.921,-52.833,-178.563,6.196,148.693
C02424=1187.200,126.672,-52.813,-178.566,6.194,148.693
C02425=1187.205,126.423,-52.794,-178.569,6.193,148.694
C02426=1187.210,126.173,-52.774,-178.571,6.191,148.694
C02427=1187.215,125.924,-52.754,-178.574,6.190,148.695
C02428=1187.219,125.675,-52.734,-178.577,6.189,148.695
C02429=1187.224,125.426,-52.715,-178.579,6.187,148.695
C02430=1187.228,125.177,-52.695,-178.582,6.186,148.696
C02431=1187.233,124.928,-52.675,-178.585,6.185,148.696
C02432=1187.238,124.679,-52.656,-178.587,6.183,148.697
C02433=1187.243,124.429,-52.636,-178.590,6.182,148.697
C02434=1187.248,124.180,-52.616,-178.593,6.181,148.698
C02435=1187.252,123.931,-52.596,-178.595,6.179,148.698
C02436=1187.258,123.682,-52.577,-178.598,6.177,148.699
C02437=1187.262,123.432,-52.557,-178.601,6.177,148.699
C02438=1187.267,123.183,-52.538,-178.603,6.175,148.700
C02439=1187.272,122.934,-52.518,-178.606,6.173,148.700
C02440=1187.276,122.685,-52.499,-178.609,6.173,148.701
C02441=1187.281,122.436,-52.479,-178.611,6.171,148.701
C02442=1187.286,122.187,-52.460,-178.614,6.169,148.702
C02443=1187.291,121.937,-52.440,-178.616,6.168,148.702
C02444=1187.296,121.688,-52.420,-178.619,6.167,148.703
C02445=1187.301,121.439,-52.400,-178.621,6.166,148.703
C02446=1187.306,121.190,-52.381,-178.624,6.164,148.703
C02447=1187.310,120.940,-52.362,-178.627,6.163,148.704
C02448=1187.315,120.692,-52.342,-178.629,6.162,148.704
C02449=1187.320,120.442,-52.323,-178.632,6.160,148.705
C02450=1187.325,120.193,-52.304,-178.635,6.159,148.705
C02451=1187.330,119.944,-52.284,-178.637,6.158,148.706
C02452=1187.334,119.694,-52.265,-178.640,6.156,148.706
C02453=1187.339,119.445,-52.246,-178.643,6.155,148.707
C02454=1187.344,119.196,-52.226,-178.645,6.154,148.707
C02455=1187.349,118.946,-52.206,-178.648,6.152,148.708
C02456=1187.353,118.698,-52.188,-178.651,6.151,148.708
C02457=1187.358,118.448,-52.168,-178.653,6.150,148.709
C02458=1187.363,118.199,-52.149,-178.656,6.148,148.709
C02459=1187.368,117.950,-52.129,-178.659,6.147,148.710
C02460=1187.373,117.701,-52.110,-178.661,6.146,148.710
C02461=1187.377,117.452,-52.091,-178.664,6.145,148.711
C02462=1187.382,117.202,-52.071,-178.667,6.143,148.711
C02463=1187.387,116.953,-52.052,-178.669,6.142,148.712
C02464=1187.391,116.704,-52.033,-178.672,6.141,148.712
C02465=1187.397,116.455,-52.013,-178.675,6.139,148.713
C02466=1187.402,116.206,-51.994,-178.677,6.138,148.713
C02467=1187.406,115.957,-51.975,-178.680,6.137,148.713
C02468=1187.411,115.707,-51.955,-178.683,6.135,148.714
C02469=1187.416,115.459,-51.936,-178.685,6.134,148.714
C02470=1187.420,115.209,-51.917,-178.688,6.133,148.715
C02471=1187.425,114.959,-51.898,-178.690,6.132,148.715
C02472=1187.431,114.710,-51.879,-178.693,6.130,148.716
C02473=1187.435,114.461,-51.860,-178.696,6.129,148.717
C02474=1187.440,114.212,-51.840,-178.698,6.128,148.717
C02475=1187.445,113.963,-51.821,-178.701,6.126,148.717
C02476=1187.449,113.714,-51.802,-178.704,6.126,148.718
C02477=1187.454,113.464,-51.783,-178.706,6.124,148.718
C02478=1187.460,113.215,-51.764,-178.709,6.122,148.719
C02479=1187.464,112.966,-51.745,-178.712,6.122,148.719
C02480=1187.469,112.717,-51.725,-178.714,6.120,148.720
C02481=1187.473,112.468,-51.706,-178.717,6.119,148.720
C02482=1187.479,112.218,-51.688,-178.720,6.117,148.721
C02483=1187.483,111.968,-51.668,-178.722,6.116,148.721
C02484=1187.488,111.720,-51.649,-178.725,6.115,148.722
C02485=1187.493,111.471,-51.630,-178.728,6.113,148.722
C02486=1187.498,111.221,-51.612,-178.730,6.112,148.723
C02487=1187.503,110.972,-51.592,-178.733,6.111,148.723
C02488=1187.507,110.723,-51.573,-178.735,6.110,148.724
C02489=1187.513,110.474,-51.555,-178.738,6.109,148.724
C02490=1187.517,110.224,-51.536,-178.740,6.108,148.725
C02491=1187.522,109.975,-51.516,-178.743,6.106,148.725
C02492=1187.526,109.726,-51.498,-178.746,6.105,148.726
C02493=1187.532,109.477,-51.479,-178.748,6.104,148.726
C02494=1187.536,109.227,-51.460,-178.751,6.102,148.727
C02495=1187.541,108.978,-51.441,-178.754,6.102,148.727
C02496=1187.546,108.729,-51.423,-178.756,6.100,148.728
C02497=1187.551,108.480,-51.403,-178.759,6.099,148.728
C02498=1187.556,108.231,-51.385,-178.762,6.097,148.729
C02499=1187.560,107.981,-51.365,-178.764,6.096,148.729
C02500=1187.565,107.732,-51.347,-178.767,6.095,148.730
C02501=1187.571,107.483,-51.328,-178.770,6.093,148.730
C02502=1187.575,107.233,-51.310,-178.772,6.093,148.731
C02503=1187.581,106.965,-51.289,-178.775,6.091,148.731
C02504=1187.585,106.696,-51.269,-178.778,6.090,148.732
C02505=1187.590,106.428,-51.248,-178.780,6.089,148.732
C02506=1187.596,106.160,-51.228,-178.784,6.087,148.733
C02507=1187.600,105.911,-51.209,-178.786,6.086,148.733
C02508=1187.605,105.661,-51.191,-178.789,6.085,148.734
C02509=1187.611,105.412,-51.172,-178.792,6.083,148.734
C02510=1187.615,105.163,-51.154,-178.794,6.083,148.735
C02511=1187.620,104.914,-51.134,-178.797,6.081,148.735
C02512=1187.625,104.665,-51.116,-178.799,6.080,148.736
C02513=1187.629,104.415,-51.097,-178.802,6.079,148.736
C02514=1187.635,104.166,-51.079,-178.804,6.078,148.737
C02515=1187.640,103.917,-51.061,-178.808,6.076,148.738
C02516=1187.644,103.667,-51.042,-178.810,6.076,148.738
C02517=1187.649,103.418,-51.023,-178.812,6.074,148.738
C02518=1187.654,103.169,-51.004,-178.815,6.073,148.739
C02519=1187.658,102.919,-50.986,-178.818,6.072,148.739
C02520=1187.664,102.670,-50.968,-178.820,6.071,148.740
C02521=1187.669,102.421,-50.949,-178.823,6.069,148.740
C02522=1187.673,102.172,-50.931,-178.826,6.069,148.741
C02523=1187.678,101.923,-50.911,-178.828,6.067,148.742
C02524=1187.683,101.673,-50.893,-178.831,6.065,148.742
C02525=1187.687,101.424,-50.875,-178.834,6.065,148.743
C02526=1187.693,101.175,-50.856,-178.836,6.063,148.743
C02527=1187.698,100.926,-50.838,-178.839,6.062,148.744
C02528=1187.703,100.676,-50.820,-178.842,6.061,148.744
C02529=1187.707,100.427,-50.801,-178.844,6.060,148.745
C02530=1187.712,100.178,-50.782,-178.847,6.058,148.745
C02531=1187.717,99.928,-50.764,-178.849,6.057,148.746
C02532=1187.721,99.679,-50.746,-178.852,6.056,148.746
C02533=1187.726,99.430,-50.727,-178.855,6.055,148.747
C02534=1187.732,99.181,-50.708,-178.858,6.054,148.747
C02535=1187.737,98.931,-50.690,-178.860,6.053,148.748
C02536=1187.741,98.681,-50.672,-178.863,6.051,148.748
C02537=1187.746,98.432,-50.654,-178.865,6.050,148.749
C02538=1187.750,98.184,-50.635,-178.867,6.050,148.749
C02539=1187.756,97.934,-50.617,-178.871,6.048,148.750
C02540=1187.761,97.685,-50.599,-178.873,6.047,148.750
C02541=1187.765,97.435,-50.581,-178.876,6.046,148.751
C02542=1187.770,97.186,-50.563,-178.878,6.045,148.751
C02543=1187.775,96.938,-50.544,-178.881,6.044,148.752
C02544=1187.781,96.688,-50.525,-178.883,6.043,148.752
C02545=1187.785,96.438,-50.507,-178.887,6.041,148.753
C02546=1187.790,96.189,-50.489,-178.889,6.040,148.753
C02547=1187.795,95.940,-50.471,-178.892,6.039,148.754
C02548=1187.800,95.691,-50.453,-178.894,6.038,148.754
C02549=1187.804,95.441,-50.435,-178.897,6.036,148.755
C02550=1187.809,95.192,-50.417,-178.899,6.036,148.755
C02551=1187.814,94.942,-50.398,-178.902,6.034,148.756
C02552=1187.819,94.694,-50.379,-178.905,6.034,148.757
C02553=1187.824,94.444,-50.361,-178.907,6.032,148.757
C02554=1187.829,94.195,-50.343,-178.910,6.031,148.758
C02555=1187.834,93.946,-50.325,-178.913,6.030,148.758
C02556=1187.838,93.696,-50.307,-178.915,6.029,148.759
C02557=1187.843,93.447,-50.289,-178.918,6.028,148.759
C02558=1187.848,93.198,-50.271,-178.921,6.027,148.760
C02559=1187.853,92.949,-50.253,-178.923,6.026,148.760
C02560=1187.858,92.699,-50.235,-178.926,6.024,148.761
C02561=1187.863,92.450,-50.217,-178.928,6.023,148.761
C02562=1187.868,92.201,-50.199,-178.931,6.022,148.762
C02563=1187.872,91.951,-50.181,-178.934,6.021,148.762
C02564=1187.877,91.702,-50.163,-178.936,6.019,148.763
C02565=1187.882,91.453,-50.145,-178.939,6.019,148.763
C02566=1187.887,91.203,-50.128,-178.942,6.017,148.764
C02567=1187.892,90.954,-50.110,-178.944,6.017,148.764
C02568=1187.897,90.705,-50.092,-178.946,6.016,148.765
C02569=1187.902,90.456,-50.074,-178.950,6.014,148.765
C02570=1187.907,90.206,-50.056,-178.952,6.013,148.766
C02571=1187.911,89.956,-50.037,-178.955,6.012,148.767
C02572=1187.916,89.707,-50.019,-178.957,6.011,148.767
C02573=1187.921,89.458,-50.001,-178.960,6.010,148.768
C02574=1187.926,89.209,-49.983,-178.962,6.009,148.768
C02575=1187.931,88.959,-49.966,-178.965,6.008,148.769
C02576=1187.936,88.710,-49.948,-178.968,6.007,148.769
C02577=1187.941,88.461,-49.930,-178.970,6.006,148.770
C02578=1187.946,88.212,-49.912,-178.973,6.004,148.770
C02579=1187.950,87.962,-49.894,-178.976,6.004,148.771
C02580=1187.955,87.713,-49.876,-178.978,6.002,148.771
C02581=1187.961,87.463,-49.859,-178.981,6.001,148.772
C02582=1187.966,87.214,-49.841,-178.983,6.001,148.772
C02583=1187.970,86.965,-49.823,-178.986,5.999,148.773
C02584=1187.975,86.716,-49.805,-178.988,5.998,148.773
C02585=1187.981,86.466,-49.788,-178.992,5.997,148.774
C02586=1187.984,86.217,-49.770,-178.994,5.996,148.774
C02587=1187.989,85.967,-49.752,-178.996,5.995,148.775
C02588=1187.994,85.718,-49.734,-178.999,5.994,148.775
C02589=1187.999,85.468,-49.717,-179.002,5.993,148.776
C02590=1188.004,85.219,-49.699,-179.004,5.991,148.777
C02591=1188.009,84.970,-49.681,-179.007,5.991,148.777
C02592=1188.014,84.720,-49.664,-179.010,5.989,148.778
C02593=1188.018,84.471,-49.646,-179.012,5.989,148.778
C02594=1188.023,84.222,-49.628,-179.015,5.988,148.779
C02595=1188.029,83.972,-49.611,-179.018,5.986,148.779
C02596=1188.033,83.723,-49.593,-179.020,5.985,148.780
C02597=1188.038,83.474,-49.575,-179.023,5.984,148.780
C02598=1188.043,83.225,-49.558,-179.025,5.983,148.781
C02599=1188.048,82.975,-49.540,-179.028,5.983,148.782
C02600=1188.053,82.726,-49.522,-179.031,5.981,148.782
C02601=1188.058,82.476,-49.505,-179.033,5.980,148.783
C02602=1188.063,82.228,-49.488,-179.035,5.979,148.783
C02603=1188.068,81.979,-49.471,-179.039,5.978,148.784
C02604=1188.073,81.729,-49.453,-179.041,5.977,148.784
C02605=1188.078,81.480,-49.435,-179.044,5.976,148.785
C02606=1188.083,81.230,-49.418,-179.047,5.975,148.785
C02607=1188.088,80.962,-49.398,-179.049,5.974,148.786
C02608=1188.093,80.694,-49.380,-179.052,5.973,148.786
C02609=1188.098,80.425,-49.361,-179.055,5.972,148.787
C02610=1188.104,80.157,-49.342,-179.057,5.971,148.788
C02611=1188.109,79.907,-49.325,-179.060,5.969,148.788
C02612=1188.113,79.658,-49.308,-179.063,5.969,148.789
C02613=1188.118,79.409,-49.290,-179.065,5.968,148.789
C02614=1188.123,79.159,-49.273,-179.068,5.967,148.790
C02615=1188.128,78.910,-49.255,-179.071,5.966,148.790
C02616=1188.133,78.661,-49.238,-179.073,5.965,148.791
C02617=1188.138,78.411,-49.221,-179.076,5.963,148.791
C02618=1188.143,78.162,-49.203,-179.079,5.963,148.792
C02619=1188.147,77.912,-49.186,-179.081,5.961,148.793
C02620=1188.153,77.663,-49.169,-179.084,5.961,148.793
C02621=1188.158,77.414,-49.151,-179.086,5.960,148.794
C02622=1188.162,77.165,-49.134,-179.089,5.958,148.794
C02623=1188.167,76.915,-49.116,-179.091,5.957,148.795
C02624=1188.172,76.666,-49.100,-179.094,5.957,148.795
C02625=1188.177,76.416,-49.082,-179.097,5.955,148.796
C02626=1188.182,76.167,-49.065,-179.099,5.955,148.796
C02627=1188.186,75.917,-49.048,-179.102,5.954,148.797
C02628=1188.192,75.668,-49.031,-179.105,5.952,148.798
C02629=1188.197,75.419,-49.013,-179.107,5.952,148.798
C02630=1188.202,75.170,-48.996,-179.109,5.951,148.799
C02631=1188.207,74.920,-48.979,-179.113,5.950,148.799
C02632=1188.211,74.671,-48.962,-179.115,5.949,148.800
C02633=1188.216,74.421,-48.944,-179.117,5.948,148.800
C02634=1188.221,74.173,-48.928,-179.120,5.946,148.801
C02635=1188.226,73.923,-48.910,-179.123,5.946,148.801
C02636=1188.231,73.674,-48.893,-179.125,5.945,148.802
C02637=1188.236,73.424,-48.876,-179.128,5.944,148.802
C02638=1188.241,73.174,-48.859,-179.131,5.943,148.803
C02639=1188.246,72.926,-48.842,-179.133,5.942,148.804
C02640=1188.251,72.676,-48.825,-179.136,5.941,148.804
C02641=1188.256,72.427,-48.808,-179.138,5.940,148.805
C02642=1188.261,72.177,-48.791,-179.141,5.939,148.805
C02643=1188.265,71.928,-48.774,-179.144,5.938,148.806
C02644=1188.271,71.679,-48.756,-179.146,5.937,148.806
C02645=1188.275,71.430,-48.740,-179.149,5.937,148.807
C02646=1188.281,71.180,-48.722,-179.152,5.935,148.808
C02647=1188.285,70.930,-48.706,-179.154,5.934,148.808
C02648=1188.290,70.680,-48.689,-179.156,5.933,148.809
C02649=1188.295,70.432,-48.672,-179.160,5.932,148.809
C02650=1188.300,70.183,-48.654,-179.162,5.931,148.810
C02651=1188.305,69.933,-48.638,-179.164,5.931,148.810
C02652=1188.310,69.683,-48.620,-179.168,5.929,148.811
C02653=1188.315,69.434,-48.604,-179.170,5.928,148.811
C02654=1188.319,69.185,-48.587,-179.172,5.928,148.812
C02655=1188.325,68.935,-48.570,-179.175,5.926,148.813
C02656=1188.329,68.686,-48.553,-179.178,5.926,148.813
C02657=1188.335,68.437,-48.537,-179.180,5.925,148.814
C02658=1188.339,68.187,-48.520,-179.183,5.923,148.814
C02659=1188.344,67.938,-48.502,-179.186,5.923,148.815
C02660=1188.349,67.688,-48.485,-179.188,5.922,148.815
C02661=1188.354,67.440,-48.469,-179.190,5.921,148.816
C02662=1188.359,67.190,-48.452,-179.193,5.920,148.816
C02663=1188.364,66.940,-48.435,-179.196,5.919,148.817
C02664=1188.369,66.692,-48.419,-179.198,5.919,148.818
C02665=1188.374,66.442,-48.401,-179.201,5.917,148.818
C02666=1188.378,66.192,-48.385,-179.204,5.916,148.819
C02667=1188.384,65.943,-48.367,-179.206,5.916,148.819
C02668=1188.389,65.694,-48.351,-179.209,5.915,148.820
C02669=1188.393,65.444,-48.334,-179.211,5.913,148.820
C02670=1188.398,65.194,-48.317,-179.214,5.913,148.821
C02671=1188.404,64.946,-48.301,-179.217,5.912,148.822
C02672=1188.408,64.696,-48.285,-179.219,5.910,148.822
C02673=1188.414,64.446,-48.268,-179.222,5.910,148.823
C02674=1188.419,64.197,-48.251,-179.224,5.909,148.823
C02675=1188.423,63.948,-48.235,-179.227,5.909,148.824
C02676=1188.428,63.698,-48.218,-179.230,5.907,148.825
C02677=1188.433,63.449,-48.201,-179.232,5.906,148.825
C02678=1188.438,63.199,-48.184,-179.235,5.906,148.826
C02679=1188.442,62.950,-48.168,-179.237,5.904,148.826
C02680=1188.448,62.701,-48.151,-179.240,5.904,148.827
C02681=1188.453,62.451,-48.134,-179.243,5.903,148.827
C02682=1188.458,62.202,-48.119,-179.245,5.902,148.828
C02683=1188.463,61.953,-48.102,-179.248,5.901,148.829
C02684=1188.468,61.703,-48.085,-179.250,5.900,148.829
C02685=1188.473,61.454,-48.068,-179.253,5.899,148.830
C02686=1188.477,61.204,-48.052,-179.255,5.899,148.830
C02687=1188.482,60.954,-48.036,-179.258,5.897,148.831
C02688=1188.488,60.705,-48.019,-179.261,5.897,148.831
C02689=1188.492,60.456,-48.002,-179.263,5.896,148.832
C02690=1188.497,60.207,-47.986,-179.266,5.895,148.832
C02691=1188.502,59.958,-47.969,-179.269,5.894,148.833
C02692=1188.507,59.708,-47.954,-179.271,5.893,148.834
C02693=1188.513,59.458,-47.936,-179.274,5.892,148.834
C02694=1188.517,59.209,-47.920,-179.276,5.891,148.835
C02695=1188.522,58.960,-47.903,-179.279,5.890,148.835
C02696=1188.527,58.710,-47.887,-179.282,5.890,148.836
C02697=1188.532,58.461,-47.871,-179.284,5.889,148.836
C02698=1188.536,58.212,-47.855,-179.286,5.888,148.837
C02699=1188.543,57.962,-47.838,-179.290,5.887,148.838
C02700=1188.547,57.712,-47.822,-179.292,5.886,148.838
C02701=1188.552,57.463,-47.805,-179.294,5.885,148.839
C02702=1188.557,57.214,-47.789,-179.297,5.885,148.839
C02703=1188.561,56.964,-47.773,-179.300,5.883,148.840
C02704=1188.566,56.715,-47.756,-179.302,5.883,148.841
C02705=1188.571,56.465,-47.740,-179.305,5.882,148.841
C02706=1188.577,56.216,-47.724,-179.307,5.881,148.842
C02707=1188.582,55.967,-47.707,-179.310,5.880,148.842
C02708=1188.587,55.717,-47.691,-179.313,5.879,148.843
C02709=1188.591,55.468,-47.675,-179.315,5.879,148.844
C02710=1188.597,55.218,-47.659,-179.317,5.878,148.844
C02711=1188.601,54.950,-47.641,-179.321,5.876,148.845
C02712=1188.607,54.681,-47.624,-179.323,5.876,148.845
C02713=1188.613,54.413,-47.607,-179.326,5.875,148.846
C02714=1188.617,54.144,-47.589,-179.329,5.874,148.847
C02715=1188.623,53.895,-47.573,-179.331,5.873,148.847
C02716=1188.628,53.645,-47.556,-179.334,5.872,148.848
C02717=1188.633,53.396,-47.540,-179.337,5.871,148.848
C02718=1188.638,53.146,-47.524,-179.339,5.870,148.849
C02719=1188.643,52.897,-47.508,-179.342,5.870,148.849
C02720=1188.648,52.648,-47.492,-179.344,5.869,148.850
C02721=1188.653,52.398,-47.476,-179.347,5.868,148.851
C02722=1188.658,52.149,-47.460,-179.350,5.867,148.851
C02723=1188.663,51.899,-47.444,-179.352,5.866,148.852
C02724=1188.668,51.650,-47.427,-179.355,5.866,148.852
C02725=1188.673,51.400,-47.411,-179.357,5.865,148.853
C02726=1188.678,51.151,-47.395,-179.359,5.864,148.853
C02727=1188.683,50.901,-47.379,-179.363,5.863,148.854
C02728=1188.688,50.652,-47.363,-179.365,5.862,148.855
C02729=1188.692,50.402,-47.347,-179.367,5.861,148.855
C02730=1188.697,50.153,-47.332,-179.370,5.861,148.856
C02731=1188.702,49.905,-47.316,-179.373,5.860,148.857
C02732=1188.707,49.654,-47.300,-179.375,5.859,148.857
C02733=1188.712,49.406,-47.283,-179.378,5.858,148.858
C02734=1188.717,49.156,-47.267,-179.381,5.858,148.858
C02735=1188.722,48.906,-47.252,-179.383,5.857,148.859
C02736=1188.727,48.657,-47.235,-179.385,5.856,148.859
C02737=1188.732,48.407,-47.219,-179.388,5.855,148.860
C02738=1188.737,48.158,-47.204,-179.391,5.854,148.861
C02739=1188.742,47.908,-47.187,-179.393,5.854,148.861
C02740=1188.747,47.659,-47.172,-179.396,5.853,148.862
C02741=1188.752,47.409,-47.156,-179.398,5.852,148.862
C02742=1188.756,47.160,-47.140,-179.401,5.852,148.863
C02743=1188.762,46.911,-47.124,-179.404,5.850,148.863
C02744=1188.767,46.661,-47.108,-179.406,5.849,148.864
C02745=1188.772,46.412,-47.092,-179.409,5.849,148.865
C02746=1188.777,46.163,-47.077,-179.411,5.848,148.865
C02747=1188.782,45.913,-47.061,-179.414,5.847,148.866
C02748=1188.787,45.663,-47.045,-179.417,5.846,148.867
C02749=1188.792,45.415,-47.029,-179.419,5.845,148.867
C02750=1188.796,45.165,-47.013,-179.422,5.845,148.868
C02751=1188.802,44.915,-46.998,-179.424,5.844,148.868
C02752=1188.807,44.665,-46.982,-179.427,5.843,148.869
C02753=1188.812,44.416,-46.966,-179.429,5.843,148.870
C02754=1188.817,44.167,-46.950,-179.432,5.841,148.870
C02755=1188.821,43.917,-46.935,-179.435,5.841,148.871
C02756=1188.826,43.668,-46.919,-179.437,5.840,148.871
C02757=1188.832,43.418,-46.903,-179.440,5.840,148.872
C02758=1188.837,43.169,-46.888,-179.442,5.839,148.872
C02759=1188.842,42.919,-46.871,-179.445,5.838,148.873
C02760=1188.846,42.670,-46.856,-179.448,5.837,148.874
C02761=1188.852,42.421,-46.841,-179.450,5.836,148.874
C02762=1188.857,42.171,-46.825,-179.453,5.835,148.875
C02763=1188.862,41.921,-46.809,-179.455,5.835,148.876
C02764=1188.867,41.672,-46.794,-179.457,5.834,148.876
C02765=1188.871,41.422,-46.778,-179.460,5.834,148.877
C02766=1188.877,41.173,-46.762,-179.463,5.833,148.877
C02767=1188.882,40.923,-46.747,-179.465,5.831,148.878
C02768=1188.886,40.675,-46.731,-179.468,5.831,148.878
C02769=1188.891,40.425,-46.715,-179.471,5.830,148.879
C02770=1188.897,40.175,-46.700,-179.473,5.829,148.880
C02771=1188.901,39.926,-46.685,-179.476,5.829,148.880
C02772=1188.907,39.677,-46.669,-179.478,5.828,148.881
C02773=1188.911,39.427,-46.653,-179.480,5.828,148.881
C02774=1188.917,39.177,-46.638,-179.484,5.826,148.882
C02775=1188.922,38.928,-46.623,-179.486,5.826,148.883
C02776=1188.927,38.679,-46.607,-179.488,5.825,148.883
C02777=1188.932,38.429,-46.591,-179.491,5.824,148.884
C02778=1188.936,38.180,-46.576,-179.494,5.824,148.884
C02779=1188.942,37.930,-46.560,-179.496,5.823,148.885
C02780=1188.947,37.681,-46.545,-179.498,5.822,148.886
C02781=1188.951,37.431,-46.529,-179.501,5.822,148.886
C02782=1188.957,37.182,-46.514,-179.504,5.820,148.887
C02783=1188.961,36.933,-46.499,-179.506,5.820,148.887
C02784=1188.967,36.683,-46.483,-179.509,5.819,148.888
C02785=1188.972,36.433,-46.468,-179.512,5.819,148.889
C02786=1188.976,36.183,-46.453,-179.514,5.818,148.889
C02787=1188.982,35.934,-46.437,-179.517,5.817,148.890
C02788=1188.987,35.685,-46.422,-179.519,5.817,148.891
C02789=1188.992,35.436,-46.407,-179.521,5.816,148.891
C02790=1188.997,35.186,-46.391,-179.525,5.815,148.892
C02791=1189.001,34.936,-46.376,-179.527,5.814,148.892
C02792=1189.007,34.687,-46.360,-179.529,5.813,148.893
C02793=1189.012,34.438,-46.345,-179.532,5.813,148.893
C02794=1189.017,34.188,-46.330,-179.535,5.812,148.894
C02795=1189.022,33.938,-46.315,-179.537,5.811,148.895
C02796=1189.027,33.689,-46.300,-179.539,5.811,148.895
C02797=1189.032,33.439,-46.284,-179.542,5.810,148.896
C02798=1189.036,33.190,-46.269,-179.544,5.809,148.896
C02799=1189.042,32.941,-46.253,-179.547,5.808,148.897
C02800=1189.047,32.691,-46.239,-179.550,5.808,148.898
C02801=1189.052,32.442,-46.223,-179.553,5.807,148.898
C02802=1189.057,32.193,-46.209,-179.555,5.806,148.899
C02803=1189.062,31.942,-46.193,-179.558,5.806,148.900
C02804=1189.066,31.693,-46.178,-179.560,5.805,148.900
C02805=1189.072,31.443,-46.163,-179.562,5.804,148.901
C02806=1189.077,31.194,-46.148,-179.565,5.804,148.901
C02807=1189.082,30.945,-46.132,-179.568,5.803,148.902
C02808=1189.087,30.695,-46.118,-179.570,5.802,148.902
C02809=1189.092,30.446,-46.102,-179.572,5.802,148.903
C02810=1189.097,30.197,-46.087,-179.576,5.801,148.904
C02811=1189.102,29.947,-46.071,-179.578,5.800,148.905
C02812=1189.107,29.697,-46.057,-179.580,5.799,148.905
C02813=1189.112,29.447,-46.041,-179.583,5.799,148.906
C02814=1189.117,29.198,-46.026,-179.586,5.798,148.906
C02815=1189.123,28.929,-46.010,-179.588,5.798,148.907
C02816=1189.128,28.660,-45.994,-179.591,5.797,148.907
C02817=1189.134,28.391,-45.978,-179.594,5.796,148.908
C02818=1189.138,28.123,-45.962,-179.596,5.795,148.909
C02819=1189.143,27.873,-45.947,-179.599,5.795,148.909
C02820=1189.149,27.624,-45.932,-179.602,5.794,148.910
C02821=1189.153,27.375,-45.917,-179.604,5.793,148.911
C02822=1189.159,27.125,-45.902,-179.607,5.793,148.911
C02823=1189.164,26.876,-45.887,-179.609,5.792,148.912
C02824=1189.169,26.626,-45.873,-179.612,5.792,148.913
C02825=1189.174,26.377,-45.857,-179.614,5.791,148.913
C02826=1189.179,26.127,-45.843,-179.617,5.790,148.914
C02827=1189.184,25.878,-45.827,-179.620,5.789,148.914
C02828=1189.189,25.629,-45.812,-179.622,5.788,148.915
C02829=1189.194,25.379,-45.798,-179.625,5.788,148.916
C02830=1189.199,25.129,-45.782,-179.627,5.787,148.916
C02831=1189.204,24.880,-45.768,-179.630,5.787,148.917
C02832=1189.209,24.631,-45.753,-179.632,5.786,148.917
C02833=1189.215,24.381,-45.738,-179.635,5.785,148.918
C02834=1189.219,24.131,-45.723,-179.637,5.785,148.919
C02835=1189.224,23.881,-45.709,-179.640,5.784,148.919
C02836=1189.229,23.632,-45.693,-179.642,5.783,148.920
C02837=1189.234,23.382,-45.679,-179.645,5.783,148.921
C02838=1189.239,23.133,-45.664,-179.648,5.782,148.921
C02839=1189.244,22.883,-45.649,-179.650,5.781,148.922
C02840=1189.249,22.634,-45.634,-179.652,5.781,148.922
C02841=1189.254,22.384,-45.620,-179.655,5.780,148.923
C02842=1189.259,22.135,-45.606,-179.657,5.780,148.924
C02843=1189.265,21.886,-45.590,-179.660,5.779,148.924
C02844=1189.270,21.636,-45.576,-179.662,5.779,148.925
C02845=1189.274,21.387,-45.561,-179.665,5.778,148.926
C02846=1189.279,21.137,-45.547,-179.667,5.777,148.926
C02847=1189.285,20.888,-45.531,-179.670,5.776,148.927
C02848=1189.290,20.638,-45.517,-179.673,5.775,148.927
C02849=1189.295,20.388,-45.502,-179.675,5.775,148.928
C02850=1189.299,20.139,-45.487,-179.678,5.774,148.928
C02851=1189.305,19.889,-45.473,-179.681,5.774,148.929
C02852=1189.310,19.639,-45.458,-179.683,5.773,148.930
C02853=1189.315,19.390,-45.443,-179.685,5.772,148.930
C02854=1189.320,19.141,-45.429,-179.688,5.772,148.931
C02855=1189.325,18.891,-45.415,-179.691,5.771,148.932
C02856=1189.330,18.642,-45.399,-179.693,5.771,148.932
C02857=1189.335,18.392,-45.385,-179.695,5.770,148.933
C02858=1189.340,18.142,-45.371,-179.698,5.769,148.933
C02859=1189.345,17.893,-45.356,-179.701,5.769,148.934
C02860=1189.350,17.644,-45.342,-179.703,5.768,148.935
C02861=1189.355,17.394,-45.327,-179.706,5.768,148.935
C02862=1189.361,17.144,-45.313,-179.708,5.767,148.936
C02863=1189.365,16.895,-45.298,-179.711,5.767,148.937
C02864=1189.370,16.646,-45.283,-179.713,5.766,148.937
C02865=1189.375,16.396,-45.269,-179.716,5.765,148.938
C02866=1189.380,16.146,-45.255,-179.718,5.765,148.938
C02867=1189.385,15.897,-45.240,-179.721,5.764,148.939
C02868=1189.390,15.647,-45.225,-179.723,5.763,148.940
C02869=1189.396,15.397,-45.211,-179.726,5.763,148.940
C02870=1189.401,15.148,-45.197,-179.728,5.762,148.941
C02871=1189.406,14.899,-45.182,-179.731,5.761,148.941
C02872=1189.411,14.649,-45.167,-179.733,5.761,148.942
C02873=1189.416,14.400,-45.153,-179.736,5.761,148.943
C02874=1189.421,14.150,-45.139,-179.739,5.760,148.944
C02875=1189.426,13.900,-45.125,-179.741,5.759,148.944
C02876=1189.431,13.651,-45.110,-179.743,5.759,148.945
C02877=1189.436,13.402,-45.096,-179.746,5.758,148.945
C02878=1189.441,13.153,-45.081,-179.749,5.758,148.946
C02879=1189.446,12.903,-45.067,-179.751,5.757,148.946
C02880=1189.451,12.653,-45.053,-179.754,5.756,148.947
C02881=1189.456,12.403,-45.039,-179.756,5.756,148.948
C02882=1189.461,12.154,-45.024,-179.759,5.755,148.949
C02883=1189.467,11.904,-45.010,-179.761,5.754,148.949
C02884=1189.472,11.655,-44.995,-179.764,5.754,148.950
C02885=1189.477,11.405,-44.981,-179.766,5.754,148.950
C02886=1189.482,11.155,-44.967,-179.769,5.753,148.951
C02887=1189.487,10.905,-44.953,-179.771,5.752,148.951
C02888=1189.492,10.656,-44.939,-179.774,5.752,148.952
C02889=1189.497,10.407,-44.924,-179.776,5.751,148.953
C02890=1189.502,10.158,-44.909,-179.779,5.750,148.953
C02891=1189.507,9.908,-44.895,-179.781,5.750,148.954
C02892=1189.512,9.658,-44.881,-179.784,5.749,148.955
C02893=1189.517,9.409,-44.867,-179.787,5.749,148.955
C02894=1189.522,9.160,-44.853,-179.789,5.748,148.956
C02895=1189.526,8.910,-44.839,-179.791,5.748,148.957
C02896=1189.531,8.660,-44.825,-179.794,5.747,148.957
C02897=1189.537,8.411,-44.811,-179.797,5.747,148.958
C02898=1189.542,8.162,-44.797,-179.799,5.746,148.958
C02899=1189.547,7.911,-44.783,-179.801,5.745,148.959
C02900=1189.552,7.662,-44.769,-179.804,5.745,148.960
C02901=1189.557,7.412,-44.754,-179.807,5.744,148.960
C02902=1189.563,7.163,-44.741,-179.809,5.743,148.961
C02903=1189.568,6.913,-44.726,-179.812,5.743,148.962
C02904=1189.573,6.664,-44.712,-179.814,5.742,148.962
C02905=1189.578,6.414,-44.698,-179.817,5.742,148.963
C02906=1189.583,6.165,-44.684,-179.819,5.741,148.963
C02907=1189.588,5.915,-44.670,-179.821,5.741,148.964
C02908=1189.592,5.666,-44.656,-179.824,5.741,148.965
C02909=1189.598,5.417,-44.642,-179.826,5.740,148.965
C02910=1189.603,5.166,-44.628,-179.829,5.740,148.966
C02911=1189.608,4.917,-44.614,-179.831,5.739,148.967
C02912=1189.613,4.667,-44.600,-179.834,5.739,148.967
C02913=1189.619,4.418,-44.586,-179.837,5.738,148.968
C02914=1189.623,4.168,-44.572,-179.839,5.737,148.968
C02915=1189.628,3.919,-44.558,-179.841,5.737,148.969
C02916=1189.633,3.670,-44.544,-179.844,5.736,148.970
C02917=1189.639,3.419,-44.530,-179.847,5.736,148.970
C02918=1189.643,3.170,-44.516,-179.849,5.735,148.971
C02919=1189.649,2.900,-44.501,-179.851,5.734,148.972
C02920=1189.655,2.632,-44.487,-179.854,5.734,148.972
C02921=1189.660,2.363,-44.471,-179.857,5.733,148.973
C02922=1189.666,2.093,-44.456,-179.859,5.733,148.974
C02923=1189.671,1.843,-44.442,-179.862,5.733,148.974
C02924=1189.676,1.594,-44.429,-179.865,5.732,148.975
C02925=1189.681,1.345,-44.415,-179.867,5.732,148.976
C02926=1189.685,1.095,-44.400,-179.870,5.731,148.976
C02927=1189.691,0.845,-44.387,-179.872,5.730,148.977
C02928=1189.696,0.596,-44.374,-179.875,5.730,148.978
C02929=1189.701,0.346,-44.359,-179.878,5.729,148.978
C02930=1189.706,0.097,-44.345,-179.880,5.728,148.979
C02931=1189.711,-0.153,-44.332,-179.882,5.728,148.979
C02932=1189.717,-0.402,-44.318,-179.885,5.727,148.980
C02933=1189.721,-0.651,-44.304,-179.888,5.727,148.981
C02934=1189.726,-0.902,-44.291,-179.890,5.726,148.981
C02935=1189.732,-1.151,-44.277,-179.892,5.726,148.982
C02936=1189.736,-1.400,-44.263,-179.895,5.726,148.983
C02937=1189.741,-1.651,-44.250,-179.897,5.725,148.983
C02938=1189.747,-1.900,-44.236,-179.899,5.725,148.984
C02939=1189.752,-2.149,-44.221,-179.902,5.724,148.984
C02940=1189.757,-2.399,-44.209,-179.905,5.724,148.985
C02941=1189.762,-2.648,-44.194,-179.907,5.723,148.986
C02942=1189.767,-2.899,-44.181,-179.909,5.722,148.986
C02943=1189.772,-3.147,-44.168,-179.912,5.722,148.987
C02944=1189.777,-3.397,-44.153,-179.915,5.721,148.988
C02945=1189.783,-3.647,-44.140,-179.917,5.721,148.988
C02946=1189.787,-3.896,-44.126,-179.920,5.720,148.989
C02947=1189.793,-4.146,-44.113,-179.922,5.720,148.990
C02948=1189.798,-4.395,-44.099,-179.924,5.720,148.990
C02949=1189.802,-4.645,-44.086,-179.927,5.719,148.991
C02950=1189.808,-4.894,-44.072,-179.929,5.719,148.991
C02951=1189.813,-5.145,-44.059,-179.932,5.718,148.992
C02952=1189.818,-5.393,-44.045,-179.934,5.718,148.993
C02953=1189.823,-5.643,-44.031,-179.937,5.717,148.993
C02954=1189.829,-5.893,-44.018,-179.939,5.716,148.994
C02955=1189.833,-6.142,-44.004,-179.942,5.716,148.995
C02956=1189.839,-6.392,-43.991,-179.945,5.715,148.995
C02957=1189.843,-6.642,-43.978,-179.947,5.715,148.996
C02958=1189.848,-6.892,-43.964,-179.950,5.714,148.997
C02959=1189.854,-7.141,-43.950,-179.952,5.714,148.997
C02960=1189.859,-7.391,-43.937,-179.954,5.714,148.998
C02961=1189.864,-7.640,-43.924,-179.957,5.713,148.999
C02962=1189.869,-7.890,-43.910,-179.959,5.713,148.999
C02963=1189.874,-8.139,-43.897,-179.962,5.712,149.000
C02964=1189.879,-8.389,-43.883,-179.964,5.712,149.000
C02965=1189.885,-8.638,-43.870,-179.967,5.711,149.001
C02966=1189.889,-8.888,-43.856,-179.970,5.711,149.002
C02967=1189.895,-9.137,-43.843,-179.972,5.710,149.002
C02968=1189.900,-9.388,-43.829,-179.974,5.710,149.003
C02969=1189.905,-9.636,-43.816,-179.977,5.710,149.004
C02970=1189.910,-9.887,-43.802,-179.979,5.709,149.004
C02971=1189.915,-10.136,-43.790,-179.981,5.708,149.005
C02972=1189.920,-10.386,-43.776,-179.984,5.708,149.005
C02973=1189.925,-10.635,-43.763,-179.987,5.707,149.006
C02974=1189.930,-10.885,-43.749,-179.989,5.707,149.007
C02975=1189.935,-11.134,-43.736,-179.992,5.706,149.008
C02976=1189.941,-11.384,-43.723,-179.994,5.706,149.008
C02977=1189.945,-11.633,-43.709,-179.996,5.706,149.009
C02978=1189.951,-11.883,-43.696,-179.999,5.706,149.009
C02979=1189.956,-12.133,-43.683,179.998,5.705,149.010
C02980=1189.962,-12.382,-43.670,179.996,5.704,149.011
C02981=1189.966,-12.632,-43.656,179.994,5.704,149.011
C02982=1189.972,-12.881,-43.643,179.991,5.703,149.012
C02983=1189.976,-13.131,-43.630,179.988,5.703,149.013
C02984=1189.981,-13.380,-43.617,179.987,5.703,149.013
C02985=1189.986,-13.630,-43.603,179.984,5.702,149.014
C02986=1189.991,-13.880,-43.591,179.981,5.702,149.014
C02987=1189.997,-14.130,-43.577,179.979,5.701,149.015
C02988=1190.001,-14.379,-43.564,179.977,5.700,149.016
C02989=1190.007,-14.628,-43.550,179.974,5.700,149.016
C02990=1190.012,-14.878,-43.537,179.971,5.700,149.017
C02991=1190.017,-15.128,-43.525,179.969,5.699,149.018
C02992=1190.022,-15.377,-43.511,179.967,5.699,149.018
C02993=1190.027,-15.627,-43.498,179.964,5.699,149.019
C02994=1190.033,-15.876,-43.485,179.962,5.698,149.020
C02995=1190.037,-16.126,-43.472,179.959,5.698,149.020
C02996=1190.043,-16.376,-43.459,179.956,5.697,149.021
C02997=1190.048,-16.626,-43.446,179.954,5.696,149.021
C02998=1190.053,-16.875,-43.432,179.952,5.696,149.022
C02999=1190.058,-17.124,-43.419,179.949,5.696,149.023
C03000=1190.063,-17.374,-43.406,179.947,5.696,149.023
C03001=1190.068,-17.624,-43.394,179.945,5.695,149.024
C03002=1190.074,-17.873,-43.380,179.942,5.694,149.025
C03003=1190.079,-18.123,-43.367,179.939,5.694,149.025
C03004=1190.084,-18.373,-43.355,179.937,5.694,149.026
C03005=1190.089,-18.623,-43.341,179.935,5.693,149.026
C03006=1190.094,-18.872,-43.328,179.932,5.693,149.027
C03007=1190.099,-19.121,-43.315,179.930,5.693,149.028
C03008=1190.104,-19.371,-43.302,179.927,5.692,149.029
C03009=1190.109,-19.621,-43.289,179.924,5.692,149.029
C03010=1190.114,-19.870,-43.277,179.922,5.691,149.030
C03011=1190.120,-20.120,-43.263,179.920,5.690,149.030
C03012=1190.125,-20.370,-43.250,179.918,5.691,149.031
C03013=1190.130,-20.619,-43.238,179.915,5.690,149.032
C03014=1190.134,-20.869,-43.225,179.913,5.689,149.032
C03015=1190.140,-21.119,-43.212,179.910,5.689,149.033
C03016=1190.145,-21.368,-43.199,179.907,5.688,149.034
C03017=1190.150,-21.618,-43.186,179.905,5.688,149.034
C03018=1190.156,-21.868,-43.173,179.903,5.688,149.035
C03019=1190.161,-22.117,-43.160,179.900,5.687,149.036
C03020=1190.166,-22.366,-43.148,179.898,5.687,149.036
C03021=1190.171,-22.616,-43.135,179.895,5.687,149.037
C03022=1190.176,-22.866,-43.122,179.893,5.686,149.038
C03023=1190.181,-23.136,-43.108,179.890,5.686,149.038
C03024=1190.188,-23.405,-43.094,179.887,5.685,149.039
C03025=1190.193,-23.675,-43.080,179.885,5.685,149.040
C03026=1190.198,-23.944,-43.067,179.882,5.684,149.040
C03027=1190.204,-24.194,-43.053,179.880,5.684,149.041
C03028=1190.209,-24.443,-43.041,179.878,5.684,149.042
C03029=1190.213,-24.693,-43.028,179.875,5.683,149.042
C03030=1190.218,-24.943,-43.015,179.872,5.683,149.043
C03031=1190.223,-25.192,-43.003,179.870,5.682,149.043
C03032=1190.229,-25.442,-42.989,179.868,5.682,149.044
C03033=1190.234,-25.692,-42.977,179.865,5.682,149.045
C03034=1190.239,-25.942,-42.965,179.863,5.681,149.046
C03035=1190.244,-26.191,-42.952,179.861,5.681,149.046
C03036=1190.250,-26.440,-42.939,179.858,5.680,149.047
C03037=1190.254,-26.690,-42.926,179.855,5.680,149.047
C03038=1190.260,-26.940,-42.913,179.853,5.680,149.048
C03039=1190.265,-27.189,-42.901,179.850,5.680,149.049
C03040=1190.270,-27.439,-42.889,179.848,5.679,149.049
C03041=1190.275,-27.689,-42.876,179.846,5.678,149.050
C03042=1190.280,-27.938,-42.863,179.843,5.678,149.051
C03043=1190.285,-28.188,-42.851,179.841,5.678,149.051
C03044=1190.290,-28.437,-42.838,179.839,5.677,149.052
C03045=1190.296,-28.687,-42.826,179.836,5.677,149.053
C03046=1190.301,-28.937,-42.813,179.833,5.676,149.053
C03047=1190.306,-29.187,-42.800,179.831,5.676,149.054
C03048=1190.311,-29.436,-42.787,179.829,5.676,149.054
C03049=1190.316,-29.685,-42.775,179.827,5.675,149.055
C03050=1190.322,-29.935,-42.763,179.824,5.675,149.056
C03051=1190.326,-30.185,-42.750,179.821,5.675,149.056
C03052=1190.332,-30.435,-42.737,179.819,5.674,149.057
C03053=1190.337,-30.684,-42.725,179.817,5.674,149.058
C03054=1190.342,-30.934,-42.713,179.814,5.674,149.058
C03055=1190.347,-31.183,-42.700,179.812,5.673,149.059
C03056=1190.352,-31.433,-42.687,179.809,5.673,149.060
C03057=1190.357,-31.683,-42.675,179.807,5.673,149.060
C03058=1190.362,-31.932,-42.663,179.805,5.672,149.061
C03059=1190.367,-32.182,-42.650,179.802,5.672,149.062
C03060=1190.373,-32.432,-42.638,179.799,5.671,149.062
C03061=1190.378,-32.681,-42.626,179.797,5.670,149.063
C03062=1190.384,-32.931,-42.612,179.795,5.671,149.063
C03063=1190.389,-33.181,-42.600,179.792,5.670,149.064
C03064=1190.394,-33.431,-42.588,179.790,5.670,149.065
C03065=1190.399,-33.680,-42.575,179.788,5.669,149.065
C03066=1190.404,-33.930,-42.563,179.786,5.669,149.066
C03067=1190.409,-34.179,-42.551,179.783,5.669,149.067
C03068=1190.415,-34.428,-42.538,179.780,5.669,149.067
C03069=1190.420,-34.678,-42.526,179.778,5.668,149.068
C03070=1190.424,-34.928,-42.514,179.775,5.667,149.069
C03071=1190.429,-35.178,-42.502,179.773,5.668,149.069
C03072=1190.434,-35.427,-42.489,179.771,5.667,149.070
C03073=1190.439,-35.677,-42.477,179.768,5.667,149.071
C03074=1190.445,-35.927,-42.465,179.766,5.666,149.071
C03075=1190.450,-36.176,-42.452,179.764,5.666,149.072
C03076=1190.455,-36.426,-42.440,179.761,5.666,149.073
C03077=1190.461,-36.675,-42.428,179.758,5.665,149.073
C03078=1190.466,-36.925,-42.416,179.756,5.664,149.074
C03079=1190.471,-37.174,-42.403,179.754,5.664,149.074
C03080=1190.476,-37.425,-42.391,179.751,5.664,149.075
C03081=1190.481,-37.674,-42.378,179.749,5.664,149.076
C03082=1190.487,-37.924,-42.366,179.747,5.663,149.076
C03083=1190.492,-38.174,-42.354,179.744,5.663,149.077
C03084=1190.497,-38.424,-42.342,179.742,5.663,149.078
C03085=1190.502,-38.673,-42.329,179.739,5.663,149.078
C03086=1190.507,-38.923,-42.318,179.737,5.662,149.079
C03087=1190.512,-39.172,-42.305,179.734,5.661,149.080
C03088=1190.517,-39.422,-42.294,179.732,5.662,149.080
C03089=1190.523,-39.671,-42.281,179.730,5.661,149.081
C03090=1190.528,-39.921,-42.269,179.727,5.661,149.082
C03091=1190.533,-40.170,-42.256,179.725,5.660,149.082
C03092=1190.539,-40.420,-42.245,179.723,5.660,149.083
C03093=1190.544,-40.670,-42.233,179.720,5.660,149.084
C03094=1190.548,-40.919,-42.221,179.717,5.659,149.084
C03095=1190.554,-41.169,-42.209,179.715,5.659,149.085
C03096=1190.559,-41.418,-42.196,179.713,5.659,149.085
C03097=1190.564,-41.668,-42.184,179.710,5.658,149.086
C03098=1190.569,-41.918,-42.172,179.708,5.658,149.087
C03099=1190.575,-42.168,-42.160,179.706,5.657,149.087
C03100=1190.580,-42.417,-42.148,179.704,5.658,149.088
C03101=1190.585,-42.667,-42.136,179.701,5.657,149.089
C03102=1190.590,-42.917,-42.124,179.698,5.657,149.089
C03103=1190.596,-43.166,-42.112,179.696,5.656,149.090
C03104=1190.601,-43.416,-42.100,179.694,5.656,149.091
C03105=1190.605,-43.665,-42.088,179.691,5.656,149.091
C03106=1190.611,-43.915,-42.076,179.689,5.655,149.092
C03107=1190.616,-44.165,-42.064,179.687,5.656,149.093
C03108=1190.621,-44.415,-42.052,179.684,5.655,149.093
C03109=1190.626,-44.664,-42.041,179.682,5.654,149.094
C03110=1190.631,-44.914,-42.028,179.679,5.654,149.095
C03111=1190.637,-45.163,-42.016,179.677,5.654,149.095
C03112=1190.642,-45.413,-42.004,179.675,5.653,149.096
C03113=1190.647,-45.663,-41.993,179.672,5.653,149.096
C03114=1190.652,-45.912,-41.980,179.669,5.653,149.097
C03115=1190.657,-46.162,-41.968,179.667,5.653,149.098
C03116=1190.663,-46.412,-41.957,179.665,5.652,149.098
C03117=1190.667,-46.661,-41.945,179.663,5.652,149.099
C03118=1190.673,-46.911,-41.933,179.660,5.652,149.100
C03119=1190.678,-47.161,-41.921,179.658,5.652,149.100
C03120=1190.683,-47.411,-41.909,179.656,5.651,149.101
C03121=1190.688,-47.661,-41.898,179.653,5.650,149.102
C03122=1190.693,-47.910,-41.885,179.651,5.651,149.102
C03123=1190.699,-48.160,-41.873,179.648,5.650,149.103
C03124=1190.703,-48.410,-41.862,179.646,5.649,149.103
C03125=1190.709,-48.660,-41.850,179.643,5.649,149.104
C03126=1190.715,-48.909,-41.838,179.641,5.649,149.105
C03127=1190.720,-49.179,-41.825,179.639,5.649,149.106
C03128=1190.725,-49.449,-41.812,179.636,5.648,149.106
C03129=1190.731,-49.719,-41.800,179.633,5.648,149.107
C03130=1190.737,-49.989,-41.787,179.631,5.648,149.108
C03131=1190.742,-50.239,-41.775,179.629,5.648,149.108
C03132=1190.747,-50.489,-41.764,179.626,5.647,149.109
C03133=1190.752,-50.739,-41.752,179.624,5.647,149.110
C03134=1190.757,-50.989,-41.741,179.621,5.646,149.110
C03135=1190.763,-51.238,-41.729,179.619,5.647,149.111
C03136=1190.768,-51.487,-41.716,179.617,5.646,149.111
C03137=1190.773,-51.737,-41.705,179.614,5.645,149.112
C03138=1190.778,-51.987,-41.693,179.612,5.646,149.113
C03139=1190.784,-52.237,-41.681,179.609,5.645,149.114
C03140=1190.788,-52.486,-41.670,179.607,5.644,149.114
C03141=1190.794,-52.736,-41.658,179.605,5.645,149.115
C03142=1190.798,-52.986,-41.647,179.602,5.644,149.115
C03143=1190.804,-53.235,-41.635,179.600,5.644,149.116
C03144=1190.809,-53.485,-41.624,179.598,5.643,149.117
C03145=1190.815,-53.735,-41.612,179.596,5.643,149.117
C03146=1190.820,-53.985,-41.600,179.593,5.643,149.118
C03147=1190.825,-54.234,-41.589,179.590,5.643,149.119
C03148=1190.830,-54.484,-41.577,179.589,5.643,149.119
C03149=1190.835,-54.734,-41.566,179.586,5.642,149.120
C03150=1190.841,-54.983,-41.554,179.583,5.642,149.121
C03151=1190.845,-55.233,-41.543,179.581,5.642,149.121
C03152=1190.851,-55.483,-41.531,179.579,5.641,149.122
C03153=1190.856,-55.732,-41.520,179.576,5.641,149.123
C03154=1190.861,-55.982,-41.508,179.574,5.641,149.123
C03155=1190.866,-56.232,-41.497,179.572,5.641,149.124
C03156=1190.872,-56.481,-41.485,179.569,5.640,149.124
C03157=1190.876,-56.731,-41.474,179.567,5.640,149.125
C03158=1190.882,-56.981,-41.462,179.565,5.640,149.126
C03159=1190.887,-57.230,-41.451,179.562,5.639,149.127
C03160=1190.892,-57.480,-41.439,179.560,5.639,149.127
C03161=1190.897,-57.729,-41.428,179.558,5.639,149.128
C03162=1190.903,-57.979,-41.416,179.555,5.639,149.128
C03163=1190.907,-58.229,-41.405,179.552,5.638,149.129
C03164=1190.913,-58.479,-41.393,179.551,5.638,149.130
C03165=1190.918,-58.729,-41.382,179.548,5.638,149.130
C03166=1190.924,-58.978,-41.371,179.545,5.637,149.131
C03167=1190.929,-59.228,-41.359,179.544,5.637,149.131
C03168=1190.934,-59.478,-41.348,179.541,5.637,149.132
C03169=1190.939,-59.727,-41.336,179.539,5.636,149.133
C03170=1190.943,-59.977,-41.325,179.536,5.637,149.134
C03171=1190.949,-60.226,-41.313,179.534,5.636,149.134
C03172=1190.954,-60.476,-41.302,179.532,5.635,149.135
C03173=1190.960,-60.726,-41.291,179.530,5.636,149.135
C03174=1190.965,-60.976,-41.280,179.527,5.635,149.136
C03175=1190.971,-61.225,-41.268,179.525,5.635,149.137
C03176=1190.975,-61.475,-41.257,179.523,5.635,149.137
C03177=1190.980,-61.724,-41.246,179.520,5.635,149.138
C03178=1190.986,-61.975,-41.234,179.517,5.634,149.139
C03179=1190.991,-62.224,-41.224,179.516,5.634,149.139
C03180=1190.996,-62.474,-41.212,179.513,5.634,149.140
C03181=1191.001,-62.723,-41.200,179.510,5.633,149.141
C03182=1191.006,-62.972,-41.189,179.508,5.634,149.141
C03183=1191.012,-63.223,-41.178,179.506,5.633,149.142
C03184=1191.017,-63.472,-41.167,179.503,5.632,149.143
C03185=1191.022,-63.722,-41.156,179.501,5.633,149.143
C03186=1191.028,-63.971,-41.144,179.499,5.632,149.144
C03187=1191.033,-64.222,-41.134,179.496,5.631,149.144
C03188=1191.038,-64.472,-41.122,179.494,5.632,149.145
C03189=1191.043,-64.720,-41.111,179.492,5.631,149.146
C03190=1191.048,-64.971,-41.100,179.490,5.631,149.146
C03191=1191.054,-65.221,-41.088,179.487,5.631,149.147
C03192=1191.059,-65.470,-41.077,179.485,5.631,149.148
C03193=1191.064,-65.719,-41.066,179.482,5.630,149.148
C03194=1191.069,-65.970,-41.055,179.480,5.630,149.149
C03195=1191.074,-66.219,-41.044,179.478,5.630,149.150
C03196=1191.079,-66.468,-41.033,179.475,5.629,149.150
C03197=1191.084,-66.719,-41.022,179.474,5.629,149.151
C03198=1191.090,-66.968,-41.010,179.471,5.629,149.152
C03199=1191.095,-67.217,-40.999,179.469,5.629,149.152
C03200=1191.100,-67.468,-40.989,179.466,5.629,149.153
C03201=1191.106,-67.718,-40.977,179.464,5.628,149.153
C03202=1191.111,-67.966,-40.966,179.462,5.628,149.154
C03203=1191.116,-68.217,-40.955,179.459,5.628,149.155
C03204=1191.121,-68.466,-40.944,179.457,5.627,149.156
C03205=1191.127,-68.716,-40.933,179.455,5.627,149.156
C03206=1191.132,-68.966,-40.922,179.452,5.627,149.157
C03207=1191.137,-69.215,-40.911,179.450,5.627,149.157
C03208=1191.143,-69.465,-40.900,179.448,5.627,149.158
C03209=1191.147,-69.715,-40.889,179.445,5.626,149.159
C03210=1191.153,-69.964,-40.878,179.443,5.626,149.159
C03211=1191.158,-70.214,-40.867,179.441,5.626,149.160
C03212=1191.163,-70.464,-40.857,179.438,5.625,149.160
C03213=1191.169,-70.714,-40.845,179.436,5.626,149.161
C03214=1191.174,-70.964,-40.834,179.434,5.625,149.162
C03215=1191.179,-71.213,-40.824,179.431,5.624,149.162
C03216=1191.184,-71.462,-40.812,179.429,5.625,149.163
C03217=1191.189,-71.713,-40.801,179.427,5.624,149.164
C03218=1191.195,-71.962,-40.790,179.424,5.624,149.165
C03219=1191.200,-72.212,-40.780,179.422,5.624,149.165
C03220=1191.205,-72.461,-40.769,179.420,5.624,149.166
C03221=1191.210,-72.711,-40.758,179.418,5.624,149.166
C03222=1191.216,-72.961,-40.747,179.416,5.623,149.167
C03223=1191.221,-73.211,-40.736,179.413,5.623,149.168
C03224=1191.226,-73.461,-40.725,179.411,5.623,149.168
C03225=1191.231,-73.710,-40.714,179.408,5.623,149.169
C03226=1191.236,-73.960,-40.704,179.406,5.622,149.169
C03227=1191.241,-74.209,-40.693,179.404,5.622,149.170
C03228=1191.247,-74.460,-40.682,179.401,5.622,149.171
C03229=1191.253,-74.709,-40.671,179.400,5.622,149.171
C03230=1191.258,-74.959,-40.660,179.397,5.621,149.172
C03231=1191.263,-75.230,-40.648,179.394,5.621,149.173
C03232=1191.269,-75.500,-40.637,179.392,5.621,149.174
C03233=1191.275,-75.771,-40.625,179.389,5.621,149.174
C03234=1191.280,-76.042,-40.613,179.387,5.621,149.175
C03235=1191.286,-76.292,-40.603,179.384,5.620,149.176
C03236=1191.290,-76.542,-40.591,179.383,5.620,149.176
C03237=1191.296,-76.791,-40.581,179.380,5.620,149.177
C03238=1191.301,-77.041,-40.571,179.377,5.619,149.178
C03239=1191.306,-77.290,-40.560,179.376,5.619,149.178
C03240=1191.311,-77.540,-40.549,179.373,5.619,149.179
C03241=1191.317,-77.790,-40.539,179.371,5.619,149.179
C03242=1191.322,-78.040,-40.528,179.369,5.618,149.180
C03243=1191.327,-78.289,-40.518,179.366,5.618,149.181
C03244=1191.333,-78.540,-40.506,179.364,5.618,149.181
C03245=1191.338,-78.789,-40.495,179.361,5.618,149.182
C03246=1191.343,-79.039,-40.485,179.360,5.618,149.183
C03247=1191.349,-79.288,-40.475,179.357,5.618,149.183
C03248=1191.354,-79.538,-40.463,179.354,5.617,149.184
C03249=1191.359,-79.788,-40.453,179.353,5.617,149.184
C03250=1191.364,-80.038,-40.443,179.350,5.617,149.185
C03251=1191.369,-80.287,-40.432,179.348,5.617,149.186
C03252=1191.374,-80.537,-40.421,179.346,5.616,149.186
C03253=1191.380,-80.787,-40.411,179.343,5.616,149.187
C03254=1191.385,-81.037,-40.400,179.341,5.616,149.188
C03255=1191.390,-81.286,-40.389,179.338,5.616,149.188
C03256=1191.395,-81.536,-40.379,179.337,5.616,149.189
C03257=1191.401,-81.786,-40.369,179.334,5.615,149.190
C03258=1191.406,-82.036,-40.358,179.331,5.615,149.190
C03259=1191.411,-82.285,-40.347,179.330,5.615,149.191
C03260=1191.417,-82.534,-40.337,179.327,5.615,149.192
C03261=1191.422,-82.785,-40.326,179.325,5.615,149.192
C03262=1191.427,-83.034,-40.316,179.323,5.614,149.193
C03263=1191.432,-83.284,-40.305,179.320,5.614,149.193
C03264=1191.438,-83.533,-40.295,179.318,5.614,149.194
C03265=1191.443,-83.783,-40.284,179.316,5.613,149.195
C03266=1191.448,-84.033,-40.274,179.314,5.614,149.195
C03267=1191.453,-84.283,-40.263,179.311,5.613,149.196
C03268=1191.459,-84.533,-40.253,179.310,5.613,149.197
C03269=1191.464,-84.782,-40.243,179.307,5.613,149.197
C03270=1191.468,-85.032,-40.232,179.304,5.612,149.198
C03271=1191.474,-85.281,-40.222,179.302,5.613,149.199
C03272=1191.479,-85.531,-40.211,179.300,5.612,149.199
C03273=1191.485,-85.781,-40.201,179.298,5.612,149.200
C03274=1191.490,-86.031,-40.191,179.295,5.612,149.201
C03275=1191.495,-86.281,-40.180,179.293,5.611,149.201
C03276=1191.501,-86.530,-40.170,179.291,5.612,149.202
C03277=1191.506,-86.781,-40.160,179.288,5.611,149.202
C03278=1191.511,-87.029,-40.149,179.287,5.611,149.203
C03279=1191.516,-87.280,-40.138,179.284,5.611,149.204
C03280=1191.521,-87.529,-40.128,179.282,5.611,149.204
C03281=1191.527,-87.778,-40.118,179.280,5.610,149.205
C03282=1191.532,-88.029,-40.108,179.277,5.610,149.206
C03283=1191.537,-88.278,-40.097,179.275,5.610,149.206
C03284=1191.543,-88.528,-40.087,179.273,5.610,149.207
C03285=1191.548,-88.778,-40.077,179.271,5.610,149.207
C03286=1191.553,-89.028,-40.066,179.268,5.610,149.208
C03287=1191.558,-89.278,-40.056,179.266,5.610,149.209
C03288=1191.563,-89.527,-40.046,179.264,5.609,149.209
C03289=1191.569,-89.777,-40.036,179.261,5.609,149.210
C03290=1191.574,-90.027,-40.025,179.259,5.609,149.211
C03291=1191.579,-90.276,-40.015,179.257,5.608,149.211
C03292=1191.585,-90.526,-40.005,179.255,5.609,149.212
C03293=1191.589,-90.776,-39.995,179.252,5.608,149.212
C03294=1191.595,-91.025,-39.985,179.250,5.608,149.213
C03295=1191.600,-91.275,-39.975,179.248,5.608,149.214
C03296=1191.605,-91.525,-39.964,179.246,5.607,149.214
C03297=1191.611,-91.775,-39.954,179.243,5.607,149.215
C03298=1191.616,-92.024,-39.944,179.241,5.607,149.216
C03299=1191.621,-92.274,-39.934,179.239,5.607,149.216
C03300=1191.627,-92.524,-39.923,179.236,5.607,149.217
C03301=1191.632,-92.773,-39.913,179.234,5.607,149.218
C03302=1191.637,-93.024,-39.903,179.232,5.606,149.218
C03303=1191.642,-93.273,-39.893,179.230,5.606,149.219
C03304=1191.648,-93.522,-39.883,179.227,5.606,149.220
C03305=1191.653,-93.773,-39.873,179.225,5.605,149.220
C03306=1191.658,-94.023,-39.863,179.223,5.606,149.221
C03307=1191.663,-94.272,-39.853,179.221,5.605,149.222
C03308=1191.669,-94.522,-39.843,179.219,5.605,149.222
C03309=1191.674,-94.772,-39.832,179.216,5.605,149.223
C03310=1191.680,-95.021,-39.822,179.215,5.605,149.223
C03311=1191.684,-95.271,-39.813,179.212,5.605,149.224
C03312=1191.689,-95.521,-39.802,179.209,5.604,149.225
C03313=1191.695,-95.770,-39.792,179.208,5.604,149.225
C03314=1191.701,-96.021,-39.782,179.205,5.604,149.226
C03315=1191.706,-96.270,-39.773,179.203,5.604,149.227
C03316=1191.711,-96.520,-39.762,179.201,5.603,149.227
C03317=1191.716,-96.770,-39.752,179.199,5.604,149.228
C03318=1191.721,-97.019,-39.742,179.196,5.603,149.228
C03319=1191.727,-97.268,-39.732,179.194,5.603,149.229
C03320=1191.732,-97.519,-39.722,179.192,5.603,149.230
C03321=1191.738,-97.769,-39.712,179.190,5.603,149.230
C03322=1191.743,-98.018,-39.702,179.187,5.603,149.231
C03323=1191.748,-98.267,-39.692,179.185,5.602,149.232
C03324=1191.753,-98.518,-39.682,179.183,5.602,149.232
C03325=1191.758,-98.768,-39.673,179.180,5.602,149.233
C03326=1191.764,-99.017,-39.663,179.178,5.602,149.233
C03327=1191.770,-99.267,-39.652,179.176,5.601,149.234
C03328=1191.774,-99.517,-39.642,179.174,5.602,149.235
C03329=1191.780,-99.767,-39.633,179.171,5.601,149.235
C03330=1191.785,-100.016,-39.623,179.170,5.601,149.236
C03331=1191.790,-100.266,-39.613,179.167,5.601,149.237
C03332=1191.795,-100.516,-39.603,179.165,5.601,149.237
C03333=1191.800,-100.766,-39.594,179.163,5.601,149.238
C03334=1191.806,-101.015,-39.583,179.161,5.601,149.238
C03335=1191.811,-101.287,-39.573,179.158,5.601,149.239
C03336=1191.818,-101.558,-39.562,179.155,5.600,149.240
C03337=1191.823,-101.830,-39.552,179.154,5.600,149.240
C03338=1191.829,-102.101,-39.541,179.151,5.600,149.241
C03339=1191.834,-102.351,-39.531,179.149,5.599,149.242
C03340=1191.839,-102.601,-39.522,179.147,5.599,149.242
C03341=1191.844,-102.851,-39.511,179.144,5.599,149.243
C03342=1191.850,-103.100,-39.501,179.142,5.599,149.244
C03343=1191.855,-103.350,-39.492,179.140,5.599,149.244
C03344=1191.861,-103.600,-39.482,179.138,5.599,149.245
C03345=1191.866,-103.849,-39.472,179.135,5.599,149.246
C03346=1191.871,-104.099,-39.463,179.134,5.599,149.246
C03347=1191.876,-104.349,-39.453,179.131,5.598,149.247
C03348=1191.882,-104.599,-39.443,179.129,5.598,149.247
C03349=1191.887,-104.849,-39.433,179.127,5.598,149.248
C03350=1191.892,-105.098,-39.423,179.124,5.597,149.249
C03351=1191.898,-105.348,-39.414,179.122,5.597,149.249
C03352=1191.903,-105.597,-39.404,179.120,5.597,149.250
C03353=1191.908,-105.848,-39.394,179.118,5.597,149.250
C03354=1191.913,-106.098,-39.385,179.115,5.597,149.251
C03355=1191.919,-106.347,-39.375,179.113,5.597,149.252
C03356=1191.924,-106.597,-39.366,179.111,5.596,149.252
C03357=1191.929,-106.846,-39.355,179.109,5.597,149.253
C03358=1191.935,-107.096,-39.347,179.106,5.596,149.254
C03359=1191.940,-107.346,-39.336,179.105,5.596,149.254
C03360=1191.945,-107.596,-39.327,179.102,5.596,149.255
C03361=1191.950,-107.846,-39.317,179.101,5.596,149.255
C03362=1191.955,-108.096,-39.308,179.098,5.595,149.256
C03363=1191.961,-108.345,-39.298,179.096,5.596,149.257
C03364=1191.966,-108.595,-39.289,179.094,5.595,149.257
C03365=1191.972,-108.845,-39.279,179.091,5.595,149.258
C03366=1191.977,-109.095,-39.270,179.089,5.595,149.259
C03367=1191.982,-109.344,-39.260,179.087,5.595,149.259
C03368=1191.988,-109.594,-39.251,179.085,5.595,149.260
C03369=1191.992,-109.844,-39.241,179.083,5.595,149.260
C03370=1191.998,-110.094,-39.231,179.080,5.594,149.261
C03371=1192.003,-110.343,-39.222,179.079,5.594,149.262
C03372=1192.009,-110.594,-39.212,179.076,5.594,149.262
C03373=1192.014,-110.843,-39.202,179.074,5.594,149.263
C03374=1192.019,-111.093,-39.193,179.072,5.594,149.264
C03375=1192.024,-111.342,-39.183,179.070,5.594,149.264
C03376=1192.030,-111.592,-39.174,179.067,5.593,149.265
C03377=1192.035,-111.842,-39.164,179.065,5.594,149.265
C03378=1192.040,-112.091,-39.155,179.063,5.593,149.266
C03379=1192.046,-112.342,-39.146,179.061,5.593,149.267
C03380=1192.051,-112.591,-39.136,179.058,5.593,149.267
C03381=1192.056,-112.841,-39.127,179.057,5.593,149.268
C03382=1192.062,-113.090,-39.117,179.054,5.592,149.269
C03383=1192.067,-113.340,-39.108,179.053,5.592,149.269
C03384=1192.072,-113.591,-39.098,179.050,5.592,149.270
C03385=1192.077,-113.840,-39.089,179.048,5.592,149.270
C03386=1192.082,-114.090,-39.080,179.046,5.592,149.271
C03387=1192.088,-114.340,-39.070,179.043,5.592,149.272
C03388=1192.093,-114.589,-39.061,179.041,5.591,149.272
C03389=1192.099,-114.840,-39.051,179.039,5.592,149.273
C03390=1192.104,-115.089,-39.042,179.037,5.591,149.273
C03391=1192.109,-115.339,-39.033,179.035,5.591,149.274
C03392=1192.115,-115.589,-39.023,179.033,5.590,149.275
C03393=1192.120,-115.839,-39.014,179.031,5.591,149.275
C03394=1192.125,-116.088,-39.005,179.028,5.591,149.276
C03395=1192.131,-116.338,-38.995,179.026,5.591,149.277
C03396=1192.136,-116.588,-38.986,179.024,5.590,149.277
C03397=1192.141,-116.837,-38.977,179.022,5.590,149.278
C03398=1192.147,-117.087,-38.967,179.019,5.590,149.278
C03399=1192.152,-117.337,-38.958,179.018,5.590,149.279
C03400=1192.157,-117.586,-38.949,179.015,5.589,149.280
C03401=1192.162,-117.836,-38.940,179.013,5.590,149.280
C03402=1192.168,-118.086,-38.930,179.011,5.589,149.281
C03403=1192.173,-118.336,-38.921,179.009,5.589,149.282
C03404=1192.178,-118.585,-38.912,179.007,5.589,149.282
C03405=1192.184,-118.836,-38.902,179.004,5.589,149.283
C03406=1192.189,-119.085,-38.893,179.002,5.588,149.283
C03407=1192.194,-119.335,-38.885,179.000,5.589,149.284
C03408=1192.199,-119.585,-38.875,178.998,5.588,149.284
C03409=1192.205,-119.835,-38.865,178.996,5.588,149.285
C03410=1192.210,-120.085,-38.857,178.993,5.588,149.286
C03411=1192.215,-120.334,-38.848,178.992,5.588,149.286
C03412=1192.220,-120.584,-38.839,178.989,5.588,149.287
C03413=1192.227,-120.833,-38.829,178.987,5.588,149.288
C03414=1192.232,-121.083,-38.820,178.985,5.587,149.288
C03415=1192.237,-121.333,-38.811,178.983,5.587,149.289
C03416=1192.242,-121.583,-38.802,178.980,5.587,149.289
C03417=1192.248,-121.833,-38.793,178.979,5.587,149.290
C03418=1192.253,-122.083,-38.784,178.976,5.586,149.291
C03419=1192.258,-122.332,-38.774,178.975,5.586,149.291
C03420=1192.263,-122.582,-38.765,178.972,5.586,149.292
C03421=1192.268,-122.832,-38.756,178.970,5.586,149.293
C03422=1192.274,-123.082,-38.747,178.968,5.586,149.293
C03423=1192.279,-123.332,-38.738,178.965,5.586,149.294
C03424=1192.285,-123.581,-38.729,178.964,5.586,149.294
C03425=1192.290,-123.831,-38.720,178.961,5.586,149.295
C03426=1192.295,-124.081,-38.711,178.960,5.586,149.295
C03427=1192.301,-124.331,-38.701,178.957,5.585,149.296
C03428=1192.306,-124.580,-38.693,178.955,5.585,149.297
C03429=1192.311,-124.830,-38.684,178.953,5.585,149.297
C03430=1192.317,-125.080,-38.675,178.951,5.585,149.298
C03431=1192.322,-125.329,-38.666,178.948,5.585,149.299
C03432=1192.327,-125.579,-38.657,178.947,5.585,149.299
C03433=1192.333,-125.829,-38.648,178.944,5.584,149.300
C03434=1192.338,-126.079,-38.639,178.942,5.584,149.300
C03435=1192.343,-126.329,-38.630,178.940,5.584,149.301
C03436=1192.348,-126.579,-38.621,178.938,5.584,149.302
C03437=1192.354,-126.828,-38.612,178.936,5.583,149.302
C03438=1192.359,-127.078,-38.603,178.934,5.583,149.303
C03439=1191.938,-127.089,-38.642,178.930,5.587,149.305
C03440=1191.933,-126.839,-38.651,178.932,5.587,149.304
C03441=1191.928,-126.589,-38.660,178.934,5.587,149.304
C03442=1191.922,-126.340,-38.668,178.936,5.587,149.303
C03443=1191.916,-126.090,-38.678,178.938,5.588,149.302
C03444=1191.911,-125.840,-38.687,178.940,5.587,149.302
C03445=1191.906,-125.590,-38.696,178.942,5.588,149.301
C03446=1191.901,-125.340,-38.705,178.944,5.588,149.300
C03447=1191.895,-125.091,-38.714,178.947,5.588,149.300
C03448=1191.890,-124.841,-38.722,178.949,5.588,149.299
C03449=1191.884,-124.591,-38.732,178.951,5.589,149.299
C03450=1191.879,-124.341,-38.741,178.953,5.589,149.298
C03451=1191.874,-124.092,-38.750,178.956,5.589,149.297
C03452=1191.868,-123.842,-38.759,178.957,5.589,149.297
C03453=1191.863,-123.592,-38.768,178.960,5.589,149.296
C03454=1191.858,-123.343,-38.777,178.962,5.589,149.296
C03455=1191.852,-123.092,-38.786,178.964,5.590,149.295
C03456=1191.847,-122.843,-38.795,178.966,5.590,149.294
C03457=1191.842,-122.593,-38.804,178.969,5.590,149.294
C03458=1191.837,-122.343,-38.813,178.970,5.590,149.293
C03459=1191.832,-122.094,-38.823,178.973,5.590,149.293
C03460=1191.826,-121.843,-38.832,178.974,5.590,149.292
C03461=1191.821,-121.594,-38.841,178.977,5.591,149.291
C03462=1191.816,-121.344,-38.850,178.979,5.591,149.291
C03463=1191.810,-121.094,-38.859,178.981,5.590,149.290
C03464=1191.805,-120.844,-38.868,178.983,5.591,149.289
C03465=1191.800,-120.595,-38.878,178.985,5.591,149.289
C03466=1191.794,-120.345,-38.886,178.988,5.591,149.288
C03467=1191.789,-120.096,-38.895,178.989,5.591,149.288
C03468=1191.783,-119.845,-38.905,178.992,5.591,149.287
C03469=1191.778,-119.596,-38.914,178.994,5.591,149.287
C03470=1191.773,-119.346,-38.923,178.996,5.592,149.286
C03471=1191.768,-119.096,-38.932,178.998,5.592,149.285
C03472=1191.762,-118.846,-38.942,179.001,5.592,149.285
C03473=1191.757,-118.596,-38.951,179.002,5.592,149.284
C03474=1191.752,-118.347,-38.960,179.005,5.593,149.283
C03475=1191.747,-118.097,-38.969,179.007,5.592,149.283
C03476=1191.741,-117.847,-38.979,179.009,5.593,149.282
C03477=1191.736,-117.597,-38.988,179.011,5.593,149.281
C03478=1191.731,-117.348,-38.997,179.013,5.593,149.281
C03479=1191.725,-117.098,-39.007,179.015,5.593,149.280
C03480=1191.720,-116.848,-39.016,179.018,5.594,149.280
C03481=1191.715,-116.599,-39.025,179.020,5.593,149.279
C03482=1191.709,-116.349,-39.035,179.022,5.594,149.279
C03483=1191.704,-116.099,-39.044,179.024,5.594,149.278
C03484=1191.698,-115.849,-39.052,179.027,5.594,149.277
C03485=1191.693,-115.599,-39.063,179.028,5.594,149.277
C03486=1191.688,-115.350,-39.072,179.031,5.594,149.276
C03487=1191.683,-115.100,-39.080,179.033,5.594,149.275
C03488=1191.677,-114.850,-39.091,179.035,5.595,149.275
C03489=1191.672,-114.600,-39.100,179.037,5.595,149.274
C03490=1191.667,-114.350,-39.108,179.040,5.595,149.274
C03491=1191.661,-114.101,-39.119,179.042,5.595,149.273
C03492=1191.656,-113.851,-39.128,179.044,5.596,149.272
C03493=1191.651,-113.602,-39.137,179.046,5.595,149.272
C03494=1191.645,-113.352,-39.147,179.048,5.596,149.271
C03495=1191.641,-113.101,-39.156,179.050,5.596,149.270
C03496=1191.635,-112.852,-39.166,179.052,5.596,149.270
C03497=1191.630,-112.602,-39.175,179.054,5.596,149.269
C03498=1191.625,-112.352,-39.184,179.057,5.596,149.269
C03499=1191.619,-112.102,-39.194,179.059,5.596,149.268
C03500=1191.614,-111.853,-39.203,179.061,5.597,149.267
C03501=1191.608,-111.603,-39.213,179.063,5.597,149.267
C03502=1191.603,-111.353,-39.222,179.066,5.597,149.266
C03503=1191.598,-111.104,-39.232,179.068,5.597,149.265
C03504=1191.592,-110.854,-39.241,179.070,5.598,149.265
C03505=1191.587,-110.604,-39.250,179.072,5.597,149.264
C03506=1191.582,-110.354,-39.260,179.074,5.598,149.264
C03507=1191.576,-110.104,-39.269,179.076,5.597,149.263
C03508=1191.571,-109.855,-39.279,179.079,5.598,149.263
C03509=1191.566,-109.605,-39.288,179.081,5.598,149.262
C03510=1191.561,-109.355,-39.299,179.083,5.598,149.261
C03511=1191.555,-109.105,-39.308,179.085,5.598,149.261
C03512=1191.551,-108.856,-39.317,179.088,5.599,149.260
C03513=1191.545,-108.606,-39.327,179.089,5.599,149.259
C03514=1191.540,-108.356,-39.337,179.092,5.599,149.259
C03515=1191.534,-108.106,-39.346,179.094,5.599,149.258
C03516=1191.529,-107.857,-39.356,179.096,5.599,149.258
C03517=1191.523,-107.607,-39.365,179.098,5.599,149.257
C03518=1191.518,-107.358,-39.375,179.100,5.600,149.256
C03519=1191.513,-107.107,-39.385,179.102,5.599,149.256
C03520=1191.508,-106.857,-39.394,179.105,5.600,149.255
C03521=1191.503,-106.608,-39.404,179.107,5.601,149.254
C03522=1191.497,-106.358,-39.413,179.109,5.600,149.254
C03523=1191.492,-106.109,-39.424,179.112,5.601,149.253
C03524=1191.487,-105.859,-39.432,179.114,5.601,149.252
C03525=1191.481,-105.609,-39.443,179.116,5.601,149.252
C03526=1191.476,-105.359,-39.452,179.118,5.601,149.251
C03527=1191.471,-105.109,-39.462,179.121,5.601,149.251
C03528=1191.466,-104.860,-39.472,179.122,5.601,149.250
C03529=1191.460,-104.610,-39.481,179.125,5.602,149.249
C03530=1191.454,-104.360,-39.491,179.127,5.601,149.249
C03531=1191.449,-104.110,-39.500,179.129,5.602,149.248
C03532=1191.444,-103.860,-39.511,179.131,5.602,149.247
C03533=1191.439,-103.611,-39.521,179.134,5.602,149.247
C03534=1191.434,-103.361,-39.530,179.136,5.602,149.246
C03535=1191.429,-103.111,-39.540,179.138,5.603,149.246
C03536=1191.423,-102.862,-39.550,179.140,5.603,149.245
C03537=1191.418,-102.612,-39.559,179.143,5.603,149.244
C03538=1191.413,-102.362,-39.569,179.145,5.603,149.244
C03539=1191.407,-102.112,-39.580,179.147,5.603,149.243
C03540=1191.402,-101.840,-39.590,179.149,5.604,149.242
C03541=1191.396,-101.570,-39.600,179.152,5.603,149.242
C03542=1191.390,-101.297,-39.611,179.154,5.604,149.241
C03543=1191.385,-101.026,-39.622,179.157,5.604,149.240
C03544=1191.379,-100.776,-39.632,179.159,5.604,149.240
C03545=1191.374,-100.527,-39.641,179.161,5.605,149.239
C03546=1191.368,-100.277,-39.651,179.163,5.604,149.238
C03547=1191.364,-100.027,-39.661,179.165,5.605,149.238
C03548=1191.358,-99.777,-39.671,179.168,5.605,149.237
C03549=1191.352,-99.528,-39.681,179.170,5.605,149.237
C03550=1191.348,-99.278,-39.691,179.172,5.605,149.236
C03551=1191.343,-99.028,-39.701,179.174,5.605,149.235
C03552=1191.337,-98.778,-39.711,179.177,5.606,149.235
C03553=1191.332,-98.529,-39.720,179.179,5.606,149.234
C03554=1191.326,-98.279,-39.731,179.181,5.606,149.233
C03555=1191.321,-98.029,-39.741,179.183,5.606,149.233
C03556=1191.316,-97.779,-39.750,179.186,5.607,149.232
C03557=1191.311,-97.530,-39.760,179.187,5.607,149.232
C03558=1191.305,-97.280,-39.770,179.190,5.607,149.231
C03559=1191.301,-97.030,-39.780,179.192,5.607,149.230
C03560=1191.295,-96.781,-39.791,179.194,5.607,149.230
C03561=1191.289,-96.530,-39.800,179.196,5.607,149.229
C03562=1191.284,-96.281,-39.810,179.199,5.607,149.228
C03563=1191.279,-96.031,-39.820,179.201,5.608,149.228
C03564=1191.274,-95.781,-39.831,179.203,5.608,149.227
C03565=1191.268,-95.532,-39.841,179.206,5.608,149.226
C03566=1191.263,-95.283,-39.850,179.208,5.608,149.226
C03567=1191.258,-95.032,-39.860,179.210,5.609,149.225
C03568=1191.252,-94.782,-39.870,179.212,5.608,149.225
C03569=1191.247,-94.533,-39.881,179.215,5.609,149.224
C03570=1191.242,-94.283,-39.891,179.217,5.609,149.223
C03571=1191.237,-94.033,-39.901,179.219,5.609,149.223
C03572=1191.231,-93.784,-39.911,179.221,5.610,149.222
C03573=1191.226,-93.534,-39.921,179.224,5.609,149.221
C03574=1191.221,-93.284,-39.931,179.226,5.610,149.221
C03575=1191.216,-93.035,-39.941,179.228,5.610,149.220
C03576=1191.210,-92.785,-39.952,179.230,5.610,149.220
C03577=1191.205,-92.534,-39.962,179.232,5.610,149.219
C03578=1191.200,-92.285,-39.971,179.235,5.611,149.218
C03579=1191.194,-92.035,-39.981,179.237,5.610,149.218
C03580=1191.189,-91.785,-39.992,179.239,5.611,149.217
C03581=1191.184,-91.536,-40.002,179.242,5.611,149.216
C03582=1191.178,-91.286,-40.012,179.244,5.611,149.216
C03583=1191.174,-91.036,-40.022,179.246,5.612,149.215
C03584=1191.168,-90.787,-40.033,179.248,5.611,149.215
C03585=1191.163,-90.537,-40.043,179.251,5.612,149.214
C03586=1191.158,-90.287,-40.053,179.252,5.612,149.213
C03587=1191.152,-90.037,-40.064,179.255,5.612,149.213
C03588=1191.147,-89.788,-40.074,179.258,5.613,149.212
C03589=1191.142,-89.538,-40.084,179.259,5.613,149.211
C03590=1191.137,-89.288,-40.094,179.262,5.613,149.211
C03591=1191.131,-89.039,-40.104,179.264,5.613,149.210
C03592=1191.126,-88.788,-40.115,179.266,5.613,149.210
C03593=1191.121,-88.539,-40.125,179.268,5.613,149.209
C03594=1191.116,-88.289,-40.135,179.271,5.614,149.208
C03595=1191.111,-88.039,-40.145,179.273,5.614,149.208
C03596=1191.105,-87.790,-40.155,179.275,5.614,149.207
C03597=1191.100,-87.540,-40.167,179.278,5.614,149.206
C03598=1191.095,-87.291,-40.177,179.280,5.614,149.206
C03599=1191.089,-87.041,-40.187,179.282,5.615,149.205
C03600=1191.084,-86.791,-40.198,179.284,5.614,149.204
C03601=1191.079,-86.541,-40.208,179.286,5.615,149.204
C03602=1191.074,-86.291,-40.218,179.289,5.616,149.203
C03603=1191.068,-86.042,-40.229,179.291,5.615,149.202
C03604=1191.064,-85.792,-40.239,179.293,5.616,149.202
C03605=1191.058,-85.542,-40.249,179.295,5.616,149.201
C03606=1191.053,-85.293,-40.259,179.298,5.616,149.201
C03607=1191.048,-85.043,-40.270,179.300,5.617,149.200
C03608=1191.042,-84.793,-40.280,179.302,5.616,149.199
C03609=1191.037,-84.543,-40.291,179.305,5.617,149.199
C03610=1191.032,-84.294,-40.301,179.307,5.617,149.198
C03611=1191.026,-84.044,-40.311,179.309,5.617,149.197
C03612=1191.021,-83.794,-40.322,179.311,5.617,149.197
C03613=1191.016,-83.545,-40.333,179.314,5.618,149.196
C03614=1191.011,-83.295,-40.344,179.316,5.618,149.196
C03615=1191.005,-83.045,-40.354,179.318,5.618,149.195
C03616=1191.000,-82.795,-40.364,179.321,5.618,149.194
C03617=1190.995,-82.545,-40.375,179.323,5.618,149.194
C03618=1190.990,-82.296,-40.386,179.325,5.619,149.193
C03619=1190.984,-82.046,-40.396,179.328,5.619,149.192
C03620=1190.979,-81.796,-40.407,179.330,5.619,149.192
C03621=1190.974,-81.546,-40.417,179.332,5.619,149.191
C03622=1190.968,-81.297,-40.428,179.334,5.619,149.190
C03623=1190.963,-81.047,-40.438,179.337,5.620,149.190
C03624=1190.958,-80.798,-40.449,179.339,5.620,149.189
C03625=1190.953,-80.547,-40.459,179.341,5.620,149.188
C03626=1190.948,-80.298,-40.470,179.343,5.621,149.188
C03627=1190.943,-80.048,-40.481,179.346,5.620,149.187
C03628=1190.937,-79.799,-40.491,179.348,5.621,149.187
C03629=1190.932,-79.548,-40.501,179.350,5.621,149.186
C03630=1190.927,-79.300,-40.512,179.353,5.621,149.185
C03631=1190.922,-79.049,-40.523,179.355,5.621,149.185
C03632=1190.916,-78.800,-40.533,179.357,5.621,149.184
C03633=1190.911,-78.550,-40.544,179.359,5.622,149.183
C03634=1190.906,-78.301,-40.555,179.362,5.622,149.183
C03635=1190.901,-78.050,-40.565,179.364,5.622,149.182
C03636=1190.895,-77.801,-40.576,179.366,5.623,149.182
C03637=1190.890,-77.551,-40.587,179.369,5.623,149.181
C03638=1190.885,-77.302,-40.597,179.371,5.623,149.180
C03639=1190.880,-77.052,-40.608,179.373,5.624,149.180
C03640=1190.874,-76.802,-40.619,179.375,5.623,149.179
C03641=1190.869,-76.552,-40.630,179.378,5.624,149.178
C03642=1190.864,-76.303,-40.640,179.380,5.624,149.178
C03643=1190.859,-76.053,-40.651,179.382,5.624,149.177
C03644=1190.853,-75.782,-40.663,179.385,5.624,149.176
